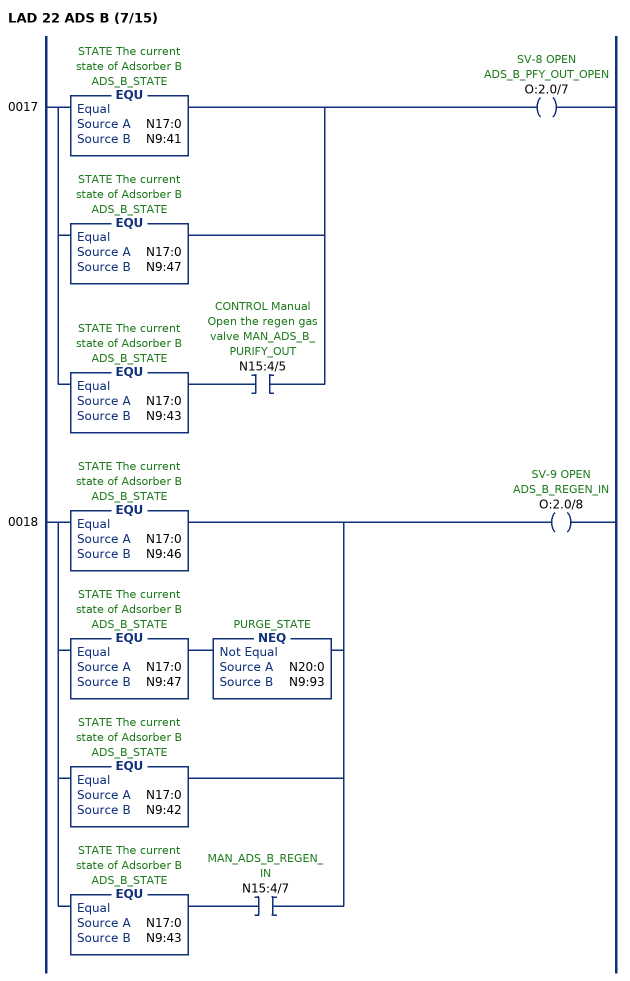
% Rung: 17 %
SOR BST EQU N17:0 N9:41 NXB EQU N17:0 N9:47 NXB EQU N17:0 N9:43 XIC N15:4/5 BND OTE O:2.0/7 EOR
%   N17:0  ADS_B_STATE  "STATE The current state of Adsorber B" %
%   N9:41  ADS_PURIFY  "STATE ADS Purify" %
%   N9:47  ADS_BACKFILL %
%   N9:43  ADS_MANUAL  "STATE ADS Manual" %
%   N15:4/5  MAN_ADS_B_PURIFY_OUT  "CONTROL Manual Open the regen gas valve" %
%   O:2.0/7  ADS_B_PFY_OUT_OPEN  "SV-8 OPEN" %
% Rung: 18 %
SOR BST EQU N17:0 N9:46 NXB EQU N17:0 N9:47 NEQ N20:0 N9:93 NXB EQU N17:0 N9:42 NXB EQU N17:0 N9:43 XIC N15:4/7 BND OTE O:2.0/8 EOR
%   N17:0  ADS_B_STATE  "STATE The current state of Adsorber B" %
%   N9:46  ADS_REGEN_BACKFILL %
%   N9:47  ADS_BACKFILL %
%   N20:0  PURGE_STATE %
%   N9:93  PURGE_BACKFILL %
%   N9:42  ADS_REGEN  "STATE ADS Regen" %
%   N9:43  ADS_MANUAL  "STATE ADS Manual" %
%   N15:4/7  MAN_ADS_B_REGEN_IN %
%   O:2.0/8  ADS_B_REGEN_IN  "SV-9 OPEN" %

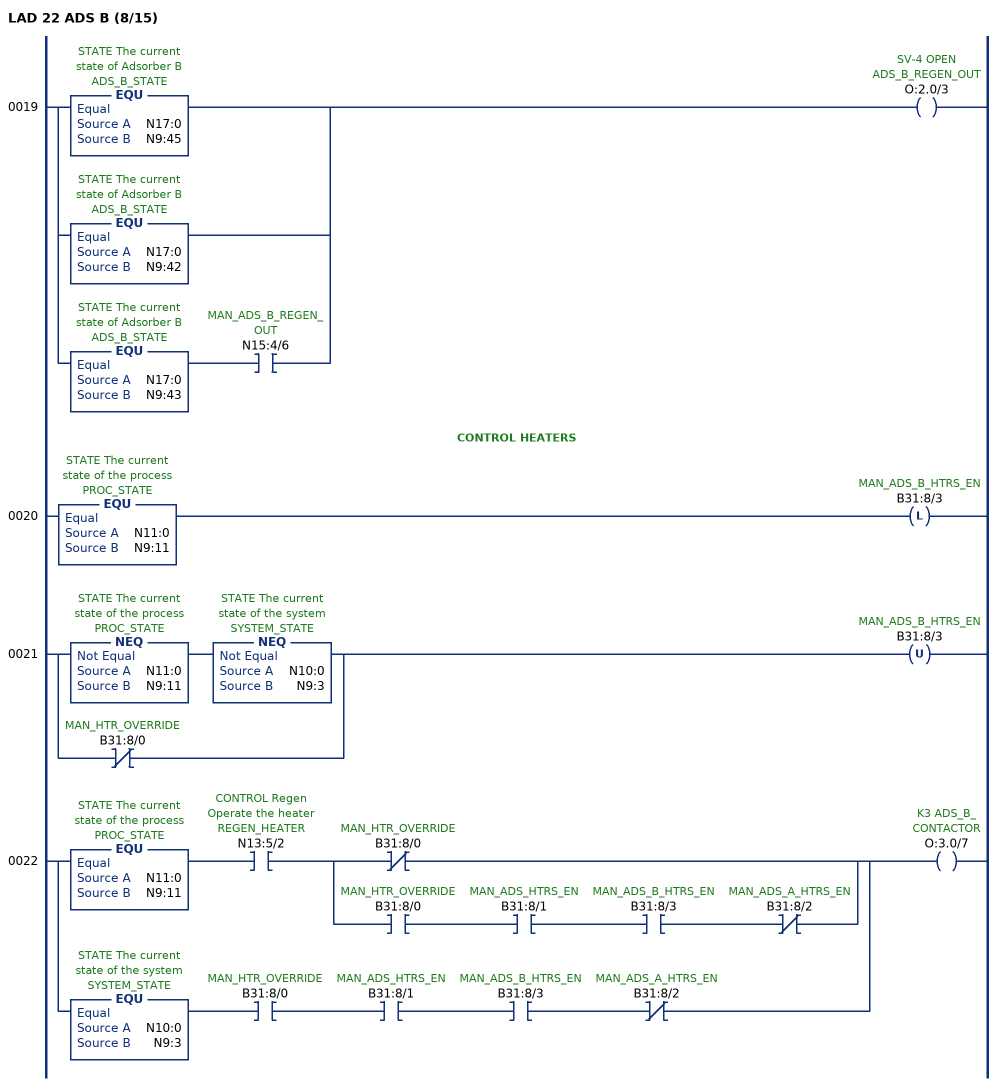
% Rung: 19 %
SOR BST EQU N17:0 N9:45 NXB EQU N17:0 N9:42 NXB EQU N17:0 N9:43 XIC N15:4/6 BND OTE O:2.0/3 EOR
%   N17:0  ADS_B_STATE  "STATE The current state of Adsorber B" %
%   N9:45  ADS_VENT %
%   N9:42  ADS_REGEN  "STATE ADS Regen" %
%   N9:43  ADS_MANUAL  "STATE ADS Manual" %
%   N15:4/6  MAN_ADS_B_REGEN_OUT %
%   O:2.0/3  ADS_B_REGEN_OUT  "SV-4 OPEN" %
% Rung: 20 %
% TITLE: CONTROL HEATERS %
SOR EQU N11:0 N9:11 OTL B31:8/3 EOR
%   N11:0  PROC_STATE  "STATE The current state of the process" %
%   N9:11  PROC_PFY_A_REG_B  "STATE Process Purify A" %
%   B31:8/3  MAN_ADS_B_HTRS_EN %
% Rung: 21 %
SOR BST NEQ N11:0 N9:11 NEQ N10:0 N9:3 NXB XIO B31:8/0 BND OTU B31:8/3 EOR
%   N11:0  PROC_STATE  "STATE The current state of the process" %
%   N9:11  PROC_PFY_A_REG_B  "STATE Process Purify A" %
%   N10:0  SYSTEM_STATE  "STATE The current state of the system" %
%   N9:3  SYSTEM_MANUAL  "STATE System Manual" %
%   B31:8/0  MAN_HTR_OVERRIDE %
%   B31:8/3  MAN_ADS_B_HTRS_EN %
% Rung: 22 %
SOR BST EQU N11:0 N9:11 XIC N13:5/2 BST XIO B31:8/0 NXB XIC B31:8/0 XIC B31:8/1 XIC B31:8/3 XIO B31:8/2 BND NXB EQU N10:0 N9:3 XIC B31:8/0 XIC B31:8/1 XIC B31:8/3 XIO B31:8/2 BND OTE O:3.0/7 EOR
%   N11:0  PROC_STATE  "STATE The current state of the process" %
%   N9:11  PROC_PFY_A_REG_B  "STATE Process Purify A" %
%   N13:5/2  REGEN_HEATER  "CONTROL Regen Operate the heater" %
%   B31:8/0  MAN_HTR_OVERRIDE %
%   B31:8/1  MAN_ADS_HTRS_EN %
%   B31:8/3  MAN_ADS_B_HTRS_EN %
%   B31:8/2  MAN_ADS_A_HTRS_EN %
%   N10:0  SYSTEM_STATE  "STATE The current state of the system" %
%   N9:3  SYSTEM_MANUAL  "STATE System Manual" %
%   O:3.0/7  ADS_B_CONTACTOR  "K3" %

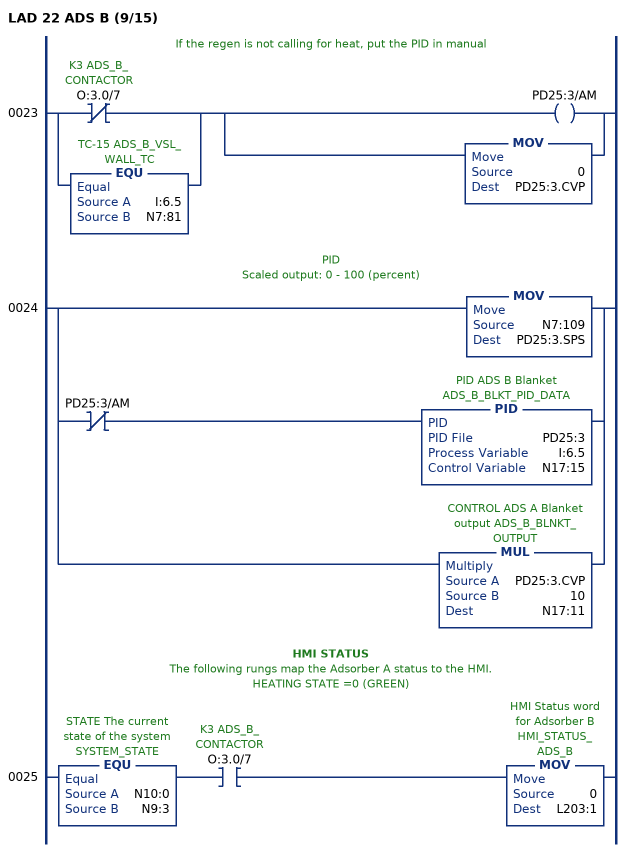
% Rung: 23 %
% If the regen is not calling for heat, put the PID in manual %
SOR BST XIO O:3.0/7 NXB EQU I:6.5 N7:81 BND BST OTE PD25:3/AM NXB MOV 0 PD25:3.CVP BND EOR
%   O:3.0/7  ADS_B_CONTACTOR  "K3" %
%   I:6.5  ADS_B_VSL_WALL_TC  "TC-15" %
%   N7:81  TC_OPEN_SP  "CONFIG The value read by an open TC input" %
% Rung: 24 %
% PID
% Scaled output: 0 - 100 (percent) %
SOR BST MOV N7:109 PD25:3.SPS NXB XIO PD25:3/AM PID PD25:3 I:6.5 N17:15 NXB MUL PD25:3.CVP 10 N17:11 BND EOR
%   N7:109  BLANKET_SP  "CONTROL Blanket PID Setpoint" %
%   PD25:3  ADS_B_BLKT_PID_DATA  "PID ADS B Blanket" %
%   I:6.5  ADS_B_VSL_WALL_TC  "TC-15" %
%   N17:15  ADS_B_BLKT_OUTPT_RAW  "CONTROL ADS B Blanket PID Output Raw" %
%   N17:11  ADS_B_BLNKT_OUTPUT  "CONTROL ADS A Blanket output" %
% Rung: 25 %
% TITLE: HMI STATUS %
% The following rungs map the Adsorber A status to the HMI.
% HEATING STATE =0 (GREEN) %
SOR EQU N10:0 N9:3 XIC O:3.0/7 MOV 0 L203:1 EOR
%   N10:0  SYSTEM_STATE  "STATE The current state of the system" %
%   N9:3  SYSTEM_MANUAL  "STATE System Manual" %
%   O:3.0/7  ADS_B_CONTACTOR  "K3" %
%   L203:1  HMI_STATUS_ADS_B  "HMI Status word for Adsorber B" %

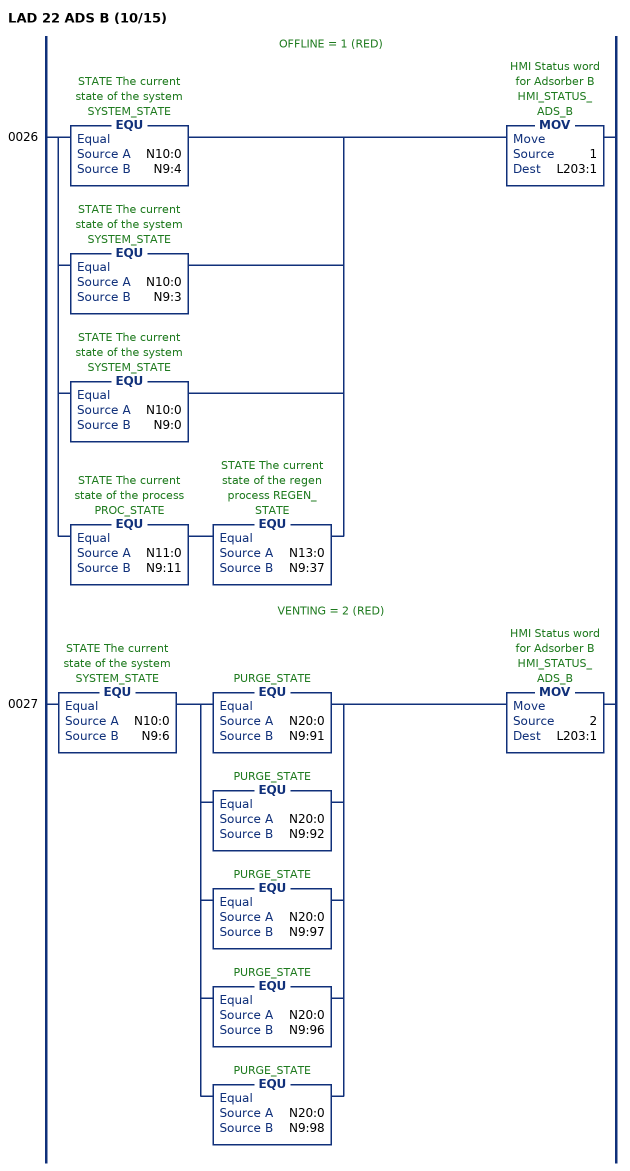
% Rung: 26 %
% OFFLINE = 1 (RED) %
SOR BST BST EQU N10:0 N9:4 NXB EQU N10:0 N9:3 NXB EQU N10:0 N9:0 BND NXB EQU N11:0 N9:11 EQU N13:0 N9:37 BND MOV 1 L203:1 EOR
%   N10:0  SYSTEM_STATE  "STATE The current state of the system" %
%   N9:4  SYSTEM_ALARM  "STATE System Alarm" %
%   N9:3  SYSTEM_MANUAL  "STATE System Manual" %
%   N9:0  SYSTEM_OFFLINE %
%   N11:0  PROC_STATE  "STATE The current state of the process" %
%   N9:11  PROC_PFY_A_REG_B  "STATE Process Purify A" %
%   N13:0  REGEN_STATE  "STATE The current state of the regen process" %
%   N9:37  REGEN_ALARM  "STATE Regen Alarm" %
%   L203:1  HMI_STATUS_ADS_B  "HMI Status word for Adsorber B" %
% Rung: 27 %
% VENTING = 2 (RED) %
SOR EQU N10:0 N9:6 BST EQU N20:0 N9:91 NXB EQU N20:0 N9:92 NXB EQU N20:0 N9:97 NXB EQU N20:0 N9:96 NXB EQU N20:0 N9:98 BND MOV 2 L203:1 EOR
%   N10:0  SYSTEM_STATE  "STATE The current state of the system" %
%   N9:6  SYSTEM_PURGE %
%   N20:0  PURGE_STATE %
%   N9:91  PURGE_INIT_VENT %
%   N9:92  PURGE_VENT_ADSORBER %
%   N9:97  PURGE_VENT_ADS_2 %
%   N9:96  PURGE_VENT_GETTER %
%   N9:98  PURGE_VENT_GET_2 %
%   L203:1  HMI_STATUS_ADS_B  "HMI Status word for Adsorber B" %

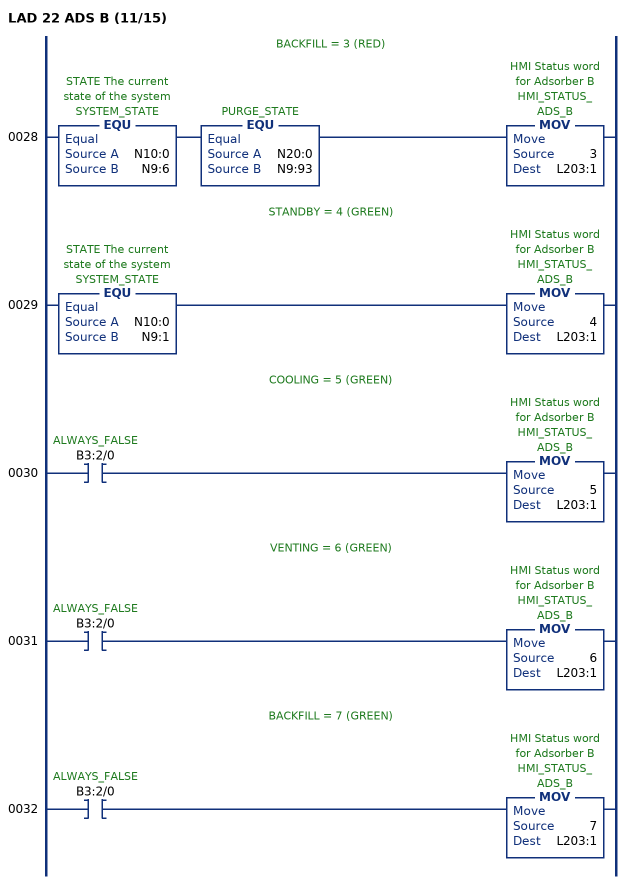
% Rung: 28 %
% BACKFILL = 3 (RED) %
SOR EQU N10:0 N9:6 EQU N20:0 N9:93 MOV 3 L203:1 EOR
%   N10:0  SYSTEM_STATE  "STATE The current state of the system" %
%   N9:6  SYSTEM_PURGE %
%   N20:0  PURGE_STATE %
%   N9:93  PURGE_BACKFILL %
%   L203:1  HMI_STATUS_ADS_B  "HMI Status word for Adsorber B" %
% Rung: 29 %
% STANDBY = 4 (GREEN) %
SOR EQU N10:0 N9:1 MOV 4 L203:1 EOR
%   N10:0  SYSTEM_STATE  "STATE The current state of the system" %
%   N9:1  SYSTEM_STANDBY  "STATE System Process" %
%   L203:1  HMI_STATUS_ADS_B  "HMI Status word for Adsorber B" %
% Rung: 30 %
% COOLING = 5 (GREEN) %
SOR XIC B3:2/0 MOV 5 L203:1 EOR
%   B3:2/0  ALWAYS_FALSE %
%   L203:1  HMI_STATUS_ADS_B  "HMI Status word for Adsorber B" %
% Rung: 31 %
% VENTING = 6 (GREEN) %
SOR XIC B3:2/0 MOV 6 L203:1 EOR
%   B3:2/0  ALWAYS_FALSE %
%   L203:1  HMI_STATUS_ADS_B  "HMI Status word for Adsorber B" %
% Rung: 32 %
% BACKFILL = 7 (GREEN) %
SOR XIC B3:2/0 MOV 7 L203:1 EOR
%   B3:2/0  ALWAYS_FALSE %
%   L203:1  HMI_STATUS_ADS_B  "HMI Status word for Adsorber B" %

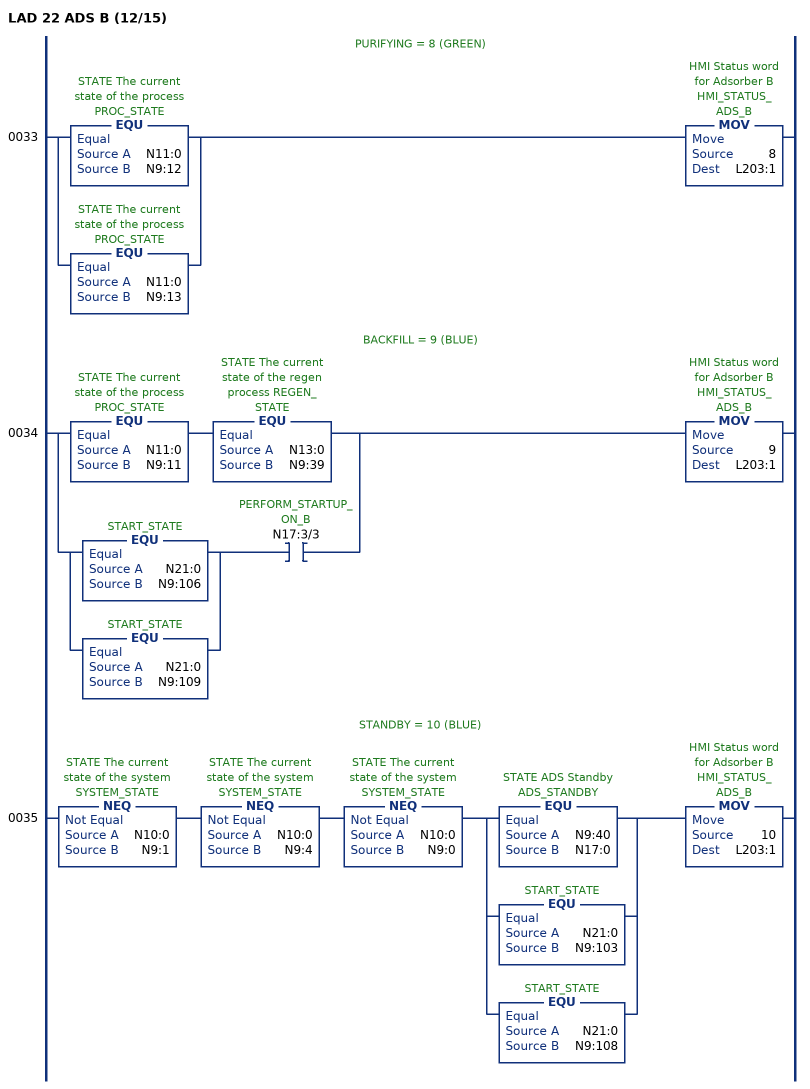
% Rung: 33 %
% PURIFYING = 8 (GREEN) %
SOR BST EQU N11:0 N9:12 NXB EQU N11:0 N9:13 BND MOV 8 L203:1 EOR
%   N11:0  PROC_STATE  "STATE The current state of the process" %
%   N9:12  PROC_PFY_B_REG_A  "STATE Process Purify B" %
%   N9:13  PROC_OVERLAP  "STATE Process Purify Overlap" %
%   L203:1  HMI_STATUS_ADS_B  "HMI Status word for Adsorber B" %
% Rung: 34 %
% BACKFILL = 9 (BLUE) %
SOR BST EQU N11:0 N9:11 EQU N13:0 N9:39 NXB BST EQU N21:0 N9:106 NXB EQU N21:0 N9:109 BND XIC N17:3/3 BND MOV 9 L203:1 EOR
%   N11:0  PROC_STATE  "STATE The current state of the process" %
%   N9:11  PROC_PFY_A_REG_B  "STATE Process Purify A" %
%   N13:0  REGEN_STATE  "STATE The current state of the regen process" %
%   N9:39  REGEN_BACKFILL %
%   N21:0  START_STATE %
%   N9:106  START_BACKFILL_1 %
%   N9:109  START_BKFL_2 %
%   N17:3/3  PERFORM_STARTUP_ON_B %
%   L203:1  HMI_STATUS_ADS_B  "HMI Status word for Adsorber B" %
% Rung: 35 %
% STANDBY = 10 (BLUE) %
SOR NEQ N10:0 N9:1 NEQ N10:0 N9:4 NEQ N10:0 N9:0 BST EQU N9:40 N17:0 NXB EQU N21:0 N9:103 NXB EQU N21:0 N9:108 BND MOV 10 L203:1 EOR
%   N10:0  SYSTEM_STATE  "STATE The current state of the system" %
%   N9:1  SYSTEM_STANDBY  "STATE System Process" %
%   N9:4  SYSTEM_ALARM  "STATE System Alarm" %
%   N9:0  SYSTEM_OFFLINE %
%   N9:40  ADS_STANDBY  "STATE ADS Standby" %
%   N17:0  ADS_B_STATE  "STATE The current state of Adsorber B" %
%   N21:0  START_STATE %
%   N9:103  START_VENT_GET_1 %
%   N9:108  START_VENT_GET_2 %
%   L203:1  HMI_STATUS_ADS_B  "HMI Status word for Adsorber B" %

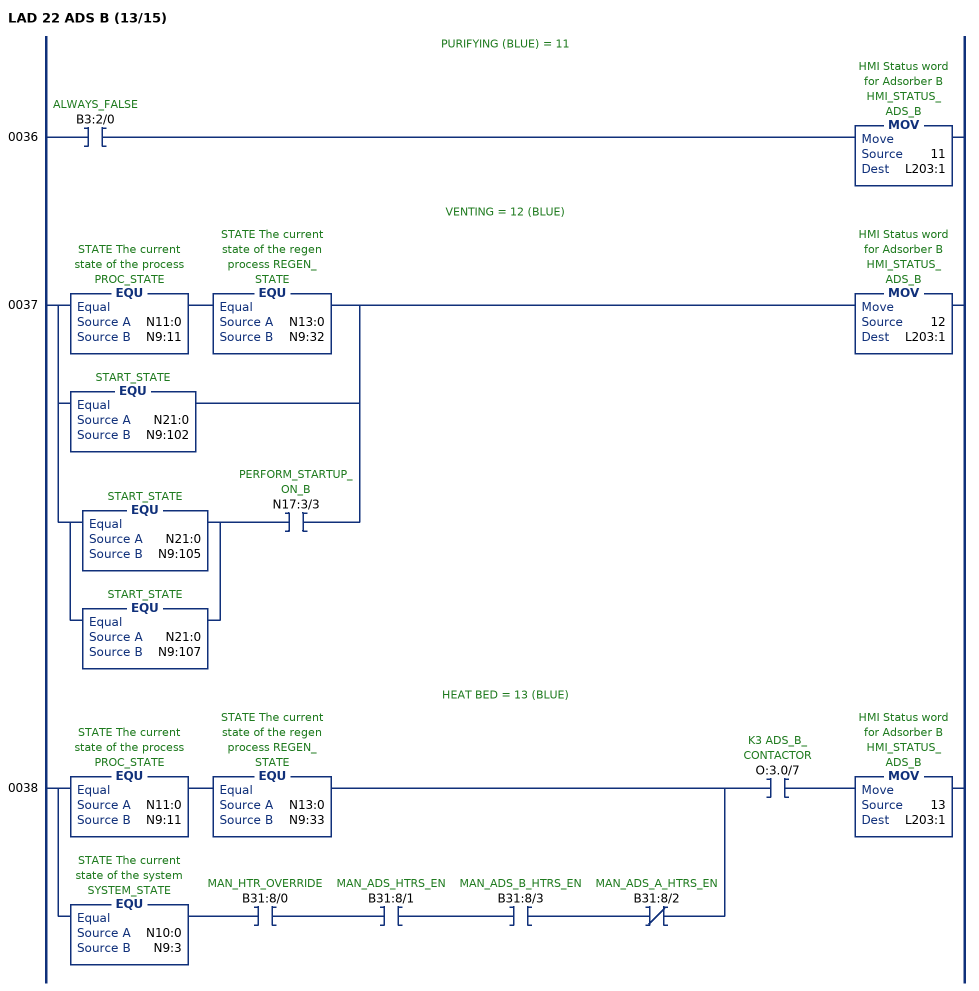
% Rung: 36 %
% PURIFYING (BLUE) = 11 %
SOR XIC B3:2/0 MOV 11 L203:1 EOR
%   B3:2/0  ALWAYS_FALSE %
%   L203:1  HMI_STATUS_ADS_B  "HMI Status word for Adsorber B" %
% Rung: 37 %
% VENTING = 12 (BLUE) %
SOR BST EQU N11:0 N9:11 EQU N13:0 N9:32 NXB BST EQU N21:0 N9:102 NXB BST EQU N21:0 N9:105 NXB EQU N21:0 N9:107 BND XIC N17:3/3 BND BND MOV 12 L203:1 EOR
%   N11:0  PROC_STATE  "STATE The current state of the process" %
%   N9:11  PROC_PFY_A_REG_B  "STATE Process Purify A" %
%   N13:0  REGEN_STATE  "STATE The current state of the regen process" %
%   N9:32  REGEN_VENT  "STATE Regen Vent" %
%   N21:0  START_STATE %
%   N9:102  START_VENT_ADS_1 %
%   N9:105  START_VENT_ALL %
%   N9:107  START_VENT_ADS_2 %
%   N17:3/3  PERFORM_STARTUP_ON_B %
%   L203:1  HMI_STATUS_ADS_B  "HMI Status word for Adsorber B" %
% Rung: 38 %
% HEAT BED = 13 (BLUE) %
SOR BST EQU N11:0 N9:11 EQU N13:0 N9:33 NXB EQU N10:0 N9:3 XIC B31:8/0 XIC B31:8/1 XIC B31:8/3 XIO B31:8/2 BND XIC O:3.0/7 MOV 13 L203:1 EOR
%   N11:0  PROC_STATE  "STATE The current state of the process" %
%   N9:11  PROC_PFY_A_REG_B  "STATE Process Purify A" %
%   N13:0  REGEN_STATE  "STATE The current state of the regen process" %
%   N9:33  REGEN_HEAT_BED  "STATE Regen Heat wall" %
%   N10:0  SYSTEM_STATE  "STATE The current state of the system" %
%   N9:3  SYSTEM_MANUAL  "STATE System Manual" %
%   B31:8/0  MAN_HTR_OVERRIDE %
%   B31:8/1  MAN_ADS_HTRS_EN %
%   B31:8/3  MAN_ADS_B_HTRS_EN %
%   B31:8/2  MAN_ADS_A_HTRS_EN %
%   O:3.0/7  ADS_B_CONTACTOR  "K3" %
%   L203:1  HMI_STATUS_ADS_B  "HMI Status word for Adsorber B" %

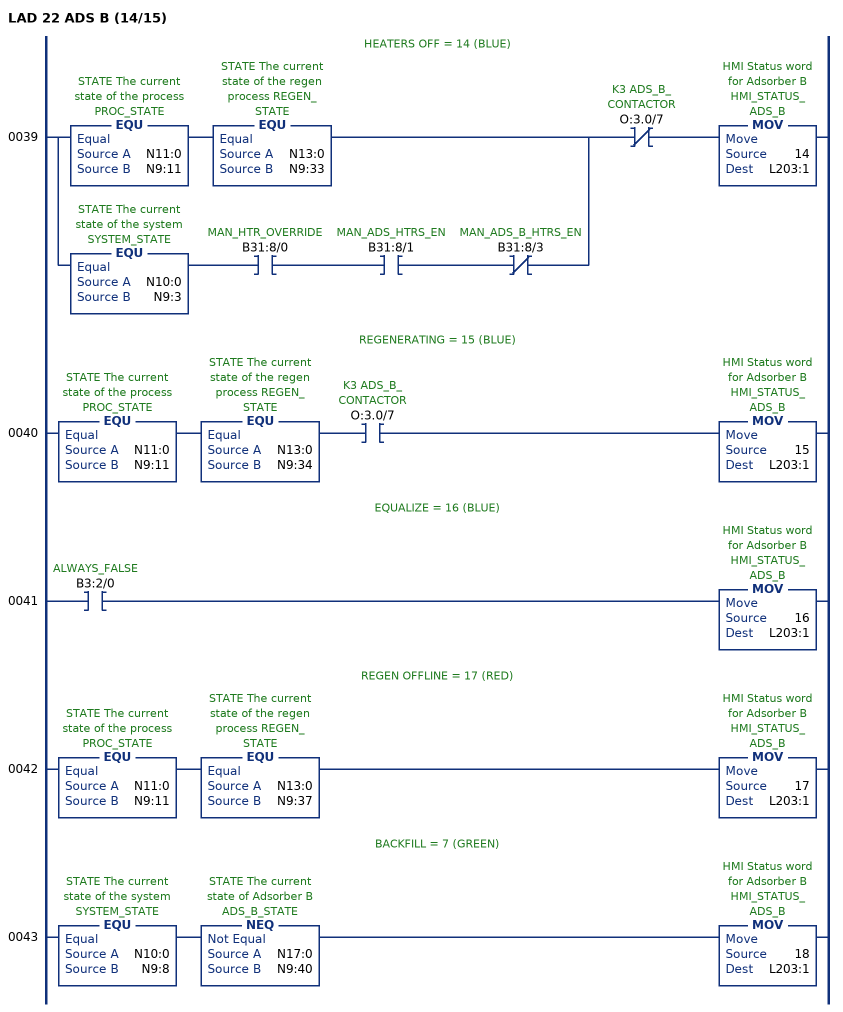
% Rung: 39 %
% HEATERS OFF = 14 (BLUE) %
SOR BST EQU N11:0 N9:11 EQU N13:0 N9:33 NXB EQU N10:0 N9:3 XIC B31:8/0 XIC B31:8/1 XIO B31:8/3 BND XIO O:3.0/7 MOV 14 L203:1 EOR
%   N11:0  PROC_STATE  "STATE The current state of the process" %
%   N9:11  PROC_PFY_A_REG_B  "STATE Process Purify A" %
%   N13:0  REGEN_STATE  "STATE The current state of the regen process" %
%   N9:33  REGEN_HEAT_BED  "STATE Regen Heat wall" %
%   N10:0  SYSTEM_STATE  "STATE The current state of the system" %
%   N9:3  SYSTEM_MANUAL  "STATE System Manual" %
%   B31:8/0  MAN_HTR_OVERRIDE %
%   B31:8/1  MAN_ADS_HTRS_EN %
%   B31:8/3  MAN_ADS_B_HTRS_EN %
%   O:3.0/7  ADS_B_CONTACTOR  "K3" %
%   L203:1  HMI_STATUS_ADS_B  "HMI Status word for Adsorber B" %
% Rung: 40 %
% REGENERATING = 15 (BLUE) %
SOR EQU N11:0 N9:11 EQU N13:0 N9:34 XIC O:3.0/7 MOV 15 L203:1 EOR
%   N11:0  PROC_STATE  "STATE The current state of the process" %
%   N9:11  PROC_PFY_A_REG_B  "STATE Process Purify A" %
%   N13:0  REGEN_STATE  "STATE The current state of the regen process" %
%   N9:34  REGEN_RUN  "STATE Regen Running" %
%   O:3.0/7  ADS_B_CONTACTOR  "K3" %
%   L203:1  HMI_STATUS_ADS_B  "HMI Status word for Adsorber B" %
% Rung: 41 %
% EQUALIZE = 16 (BLUE) %
SOR XIC B3:2/0 MOV 16 L203:1 EOR
%   B3:2/0  ALWAYS_FALSE %
%   L203:1  HMI_STATUS_ADS_B  "HMI Status word for Adsorber B" %
% Rung: 42 %
% REGEN OFFLINE = 17 (RED) %
SOR EQU N11:0 N9:11 EQU N13:0 N9:37 MOV 17 L203:1 EOR
%   N11:0  PROC_STATE  "STATE The current state of the process" %
%   N9:11  PROC_PFY_A_REG_B  "STATE Process Purify A" %
%   N13:0  REGEN_STATE  "STATE The current state of the regen process" %
%   N9:37  REGEN_ALARM  "STATE Regen Alarm" %
%   L203:1  HMI_STATUS_ADS_B  "HMI Status word for Adsorber B" %
% Rung: 43 %
% BACKFILL = 7 (GREEN) %
SOR EQU N10:0 N9:8 NEQ N17:0 N9:40 MOV 18 L203:1 EOR
%   N10:0  SYSTEM_STATE  "STATE The current state of the system" %
%   N9:8  SYSTEM_SUPPLEMENTAL %
%   N17:0  ADS_B_STATE  "STATE The current state of Adsorber B" %
%   N9:40  ADS_STANDBY  "STATE ADS Standby" %
%   L203:1  HMI_STATUS_ADS_B  "HMI Status word for Adsorber B" %

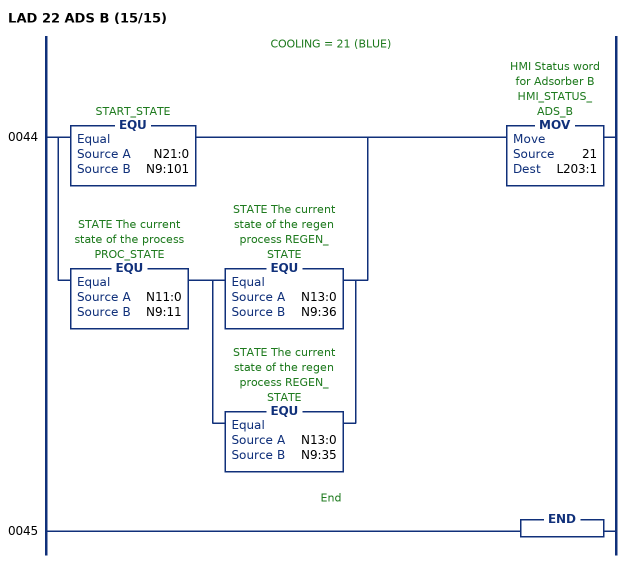
% Rung: 44 %
% COOLING = 21 (BLUE) %
SOR BST EQU N21:0 N9:101 NXB EQU N11:0 N9:11 BST EQU N13:0 N9:36 NXB EQU N13:0 N9:35 BND BND MOV 21 L203:1 EOR
%   N21:0  START_STATE %
%   N9:101  START_COOL %
%   N11:0  PROC_STATE  "STATE The current state of the process" %
%   N9:11  PROC_PFY_A_REG_B  "STATE Process Purify A" %
%   N13:0  REGEN_STATE  "STATE The current state of the regen process" %
%   N9:36  REGEN_COOL  "STATE Regen Cool" %
%   N9:35  REGEN_COOL_WALL  "STATE Regen Cool wall" %
%   L203:1  HMI_STATUS_ADS_B  "HMI Status word for Adsorber B" %
% Rung: 45 %
% End %
SOR END EOR

LADDER 23 "ADS B FLT"    % Controls the Adsorber B faults %
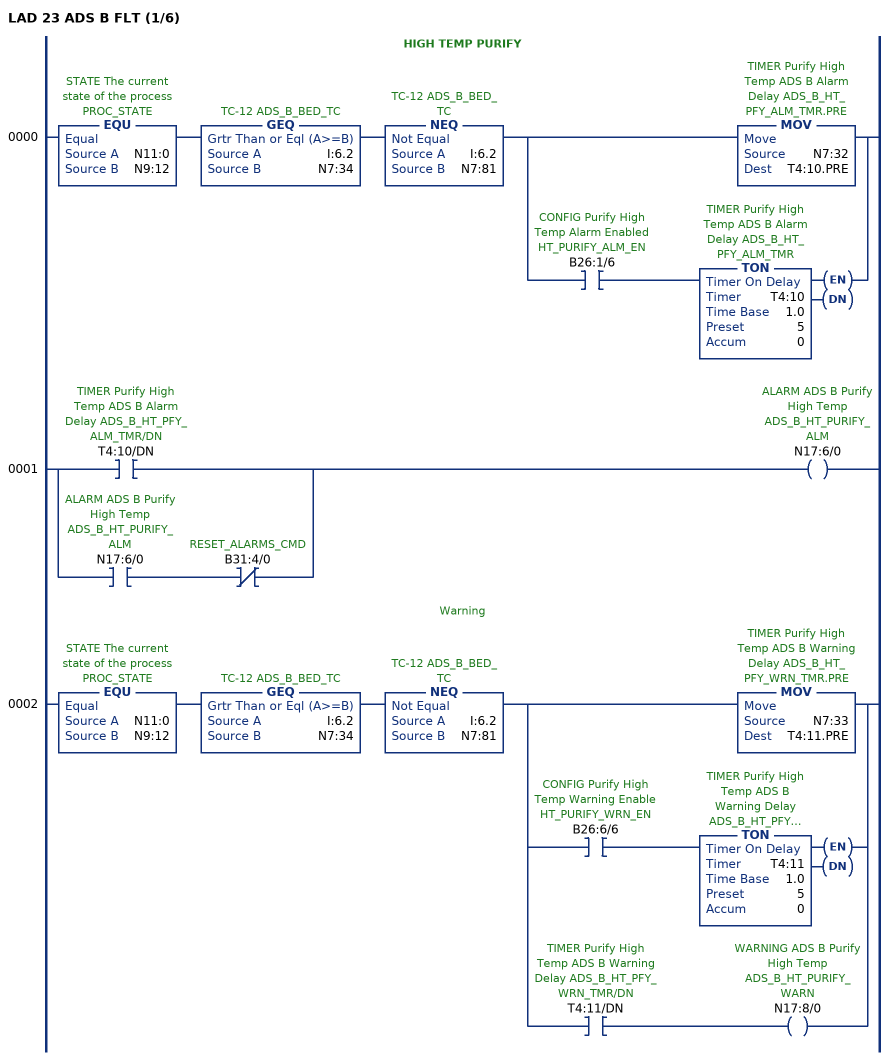
% Rung: 0 %
% TITLE: HIGH TEMP PURIFY %
SOR EQU N11:0 N9:12 GEQ I:6.2 N7:34 NEQ I:6.2 N7:81 BST MOV N7:32 T4:10.PRE NXB XIC B26:1/6 TON T4:10 1.0 5 0 BND EOR
%   N11:0  PROC_STATE  "STATE The current state of the process" %
%   N9:12  PROC_PFY_B_REG_A  "STATE Process Purify B" %
%   I:6.2  ADS_B_BED_TC  "TC-12" %
%   N7:34  HT_PURIFY_ALM_SP  "CONFIG Purify High Temp Alarm Setpoint" %
%   N7:81  TC_OPEN_SP  "CONFIG The value read by an open TC input" %
%   N7:32  HT_PURIFY_ALM_DLY  "CONFIG Purify High Temp Alarm Delay" %
%   T4:10  ADS_B_HT_PFY_ALM_TMR  "TIMER Purify High Temp ADS B Alarm Delay" %
%   B26:1/6  HT_PURIFY_ALM_EN  "CONFIG Purify High Temp Alarm Enabled" %
% Rung: 1 %
SOR BST XIC T4:10/DN NXB XIC N17:6/0 XIO B31:4/0 BND OTE N17:6/0 EOR
%   T4:10  ADS_B_HT_PFY_ALM_TMR  "TIMER Purify High Temp ADS B Alarm Delay" %
%   N17:6/0  ADS_B_HT_PURIFY_ALM  "ALARM ADS B Purify High Temp" %
%   B31:4/0  RESET_ALARMS_CMD %
% Rung: 2 %
% Warning %
SOR EQU N11:0 N9:12 GEQ I:6.2 N7:34 NEQ I:6.2 N7:81 BST MOV N7:33 T4:11.PRE NXB XIC B26:6/6 TON T4:11 1.0 5 0 NXB XIC T4:11/DN OTE N17:8/0 BND EOR
%   N11:0  PROC_STATE  "STATE The current state of the process" %
%   N9:12  PROC_PFY_B_REG_A  "STATE Process Purify B" %
%   I:6.2  ADS_B_BED_TC  "TC-12" %
%   N7:34  HT_PURIFY_ALM_SP  "CONFIG Purify High Temp Alarm Setpoint" %
%   N7:81  TC_OPEN_SP  "CONFIG The value read by an open TC input" %
%   N7:33  HT_PURIFY_WRN_DLY  "CONFIG Purify High Temp Warning Delay" %
%   T4:11  ADS_B_HT_PFY_WRN_TMR  "TIMER Purify High Temp ADS B Warning Delay" %
%   B26:6/6  HT_PURIFY_WRN_EN  "CONFIG Purify High Temp Warning Enable" %
%   N17:8/0  ADS_B_HT_PURIFY_WARN  "WARNING ADS B Purify High Temp" %

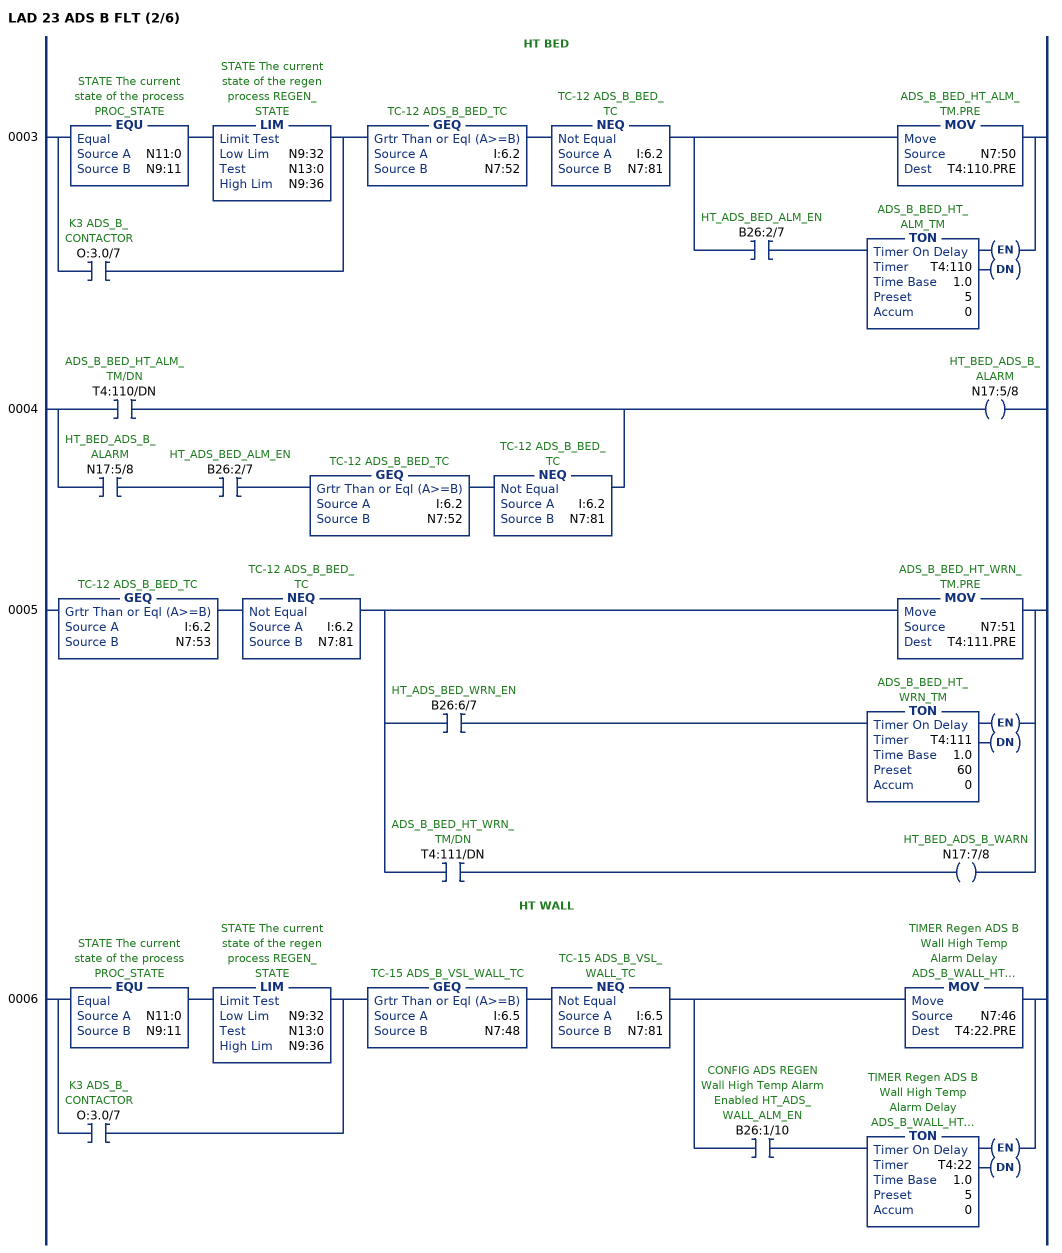
% Rung: 3 %
% TITLE: HT BED %
SOR BST EQU N11:0 N9:11 LIM N9:32 N13:0 N9:36 NXB XIC O:3.0/7 BND GEQ I:6.2 N7:52 NEQ I:6.2 N7:81 BST MOV N7:50 T4:110.PRE NXB XIC B26:2/7 TON T4:110 1.0 5 0 BND EOR
%   N11:0  PROC_STATE  "STATE The current state of the process" %
%   N9:11  PROC_PFY_A_REG_B  "STATE Process Purify A" %
%   N9:32  REGEN_VENT  "STATE Regen Vent" %
%   N13:0  REGEN_STATE  "STATE The current state of the regen process" %
%   N9:36  REGEN_COOL  "STATE Regen Cool" %
%   O:3.0/7  ADS_B_CONTACTOR  "K3" %
%   I:6.2  ADS_B_BED_TC  "TC-12" %
%   N7:52  HT_ADS_BED_ALM_SP %
%   N7:81  TC_OPEN_SP  "CONFIG The value read by an open TC input" %
%   N7:50  HT_ADS_BED_ALM_DLY %
%   T4:110  ADS_B_BED_HT_ALM_TM %
%   B26:2/7  HT_ADS_BED_ALM_EN %
% Rung: 4 %
SOR BST XIC T4:110/DN NXB XIC N17:5/8 XIC B26:2/7 GEQ I:6.2 N7:52 NEQ I:6.2 N7:81 BND OTE N17:5/8 EOR
%   T4:110  ADS_B_BED_HT_ALM_TM %
%   N17:5/8  HT_BED_ADS_B_ALARM %
%   B26:2/7  HT_ADS_BED_ALM_EN %
%   I:6.2  ADS_B_BED_TC  "TC-12" %
%   N7:52  HT_ADS_BED_ALM_SP %
%   N7:81  TC_OPEN_SP  "CONFIG The value read by an open TC input" %
% Rung: 5 %
SOR GEQ I:6.2 N7:53 NEQ I:6.2 N7:81 BST MOV N7:51 T4:111.PRE NXB XIC B26:6/7 TON T4:111 1.0 60 0 NXB XIC T4:111/DN OTE N17:7/8 BND EOR
%   I:6.2  ADS_B_BED_TC  "TC-12" %
%   N7:53  HT_ADS_BED_WRN_SP %
%   N7:81  TC_OPEN_SP  "CONFIG The value read by an open TC input" %
%   N7:51  HT_ADS_BED_WRN_DLY %
%   T4:111  ADS_B_BED_HT_WRN_TM %
%   B26:6/7  HT_ADS_BED_WRN_EN %
%   N17:7/8  HT_BED_ADS_B_WARN %
% Rung: 6 %
% TITLE: HT WALL %
SOR BST EQU N11:0 N9:11 LIM N9:32 N13:0 N9:36 NXB XIC O:3.0/7 BND GEQ I:6.5 N7:48 NEQ I:6.5 N7:81 BST MOV N7:46 T4:22.PRE NXB XIC B26:1/10 TON T4:22 1.0 5 0 BND EOR
%   N11:0  PROC_STATE  "STATE The current state of the process" %
%   N9:11  PROC_PFY_A_REG_B  "STATE Process Purify A" %
%   N9:32  REGEN_VENT  "STATE Regen Vent" %
%   N13:0  REGEN_STATE  "STATE The current state of the regen process" %
%   N9:36  REGEN_COOL  "STATE Regen Cool" %
%   O:3.0/7  ADS_B_CONTACTOR  "K3" %
%   I:6.5  ADS_B_VSL_WALL_TC  "TC-15" %
%   N7:48  HT_ADS_WALL_ALM_SP  "CONFIG ADS Wall Regen High Temp Alarm" %
%   N7:81  TC_OPEN_SP  "CONFIG The value read by an open TC input" %
%   N7:46  HT_ADS_WALL_ALM_DLY  "CONFIG ADS Wall High Temperature Alarm Delay" %
%   T4:22  ADS_B_WALL_HT_ALM_TM  "TIMER Regen ADS B Wall High Temp Alarm Delay" %
%   B26:1/10  HT_ADS_WALL_ALM_EN  "CONFIG ADS REGEN Wall High Temp Alarm Enabled" %

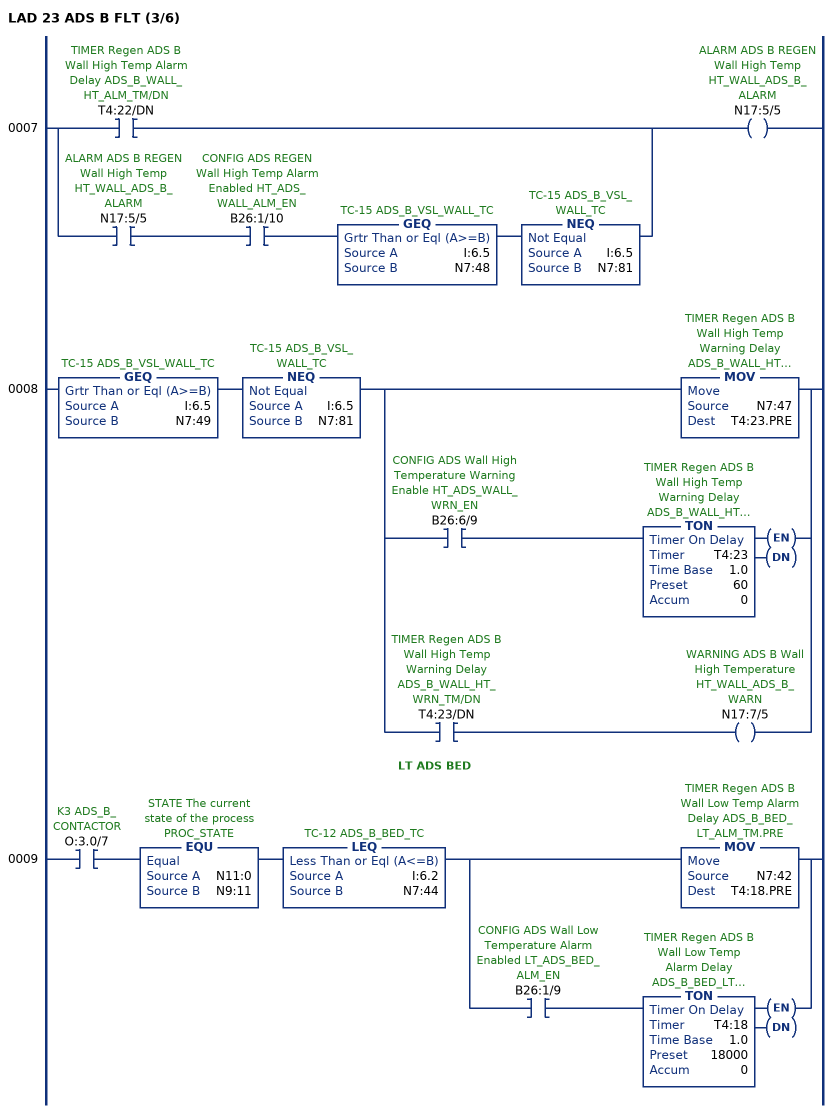
% Rung: 7 %
SOR BST XIC T4:22/DN NXB XIC N17:5/5 XIC B26:1/10 GEQ I:6.5 N7:48 NEQ I:6.5 N7:81 BND OTE N17:5/5 EOR
%   T4:22  ADS_B_WALL_HT_ALM_TM  "TIMER Regen ADS B Wall High Temp Alarm Delay" %
%   N17:5/5  HT_WALL_ADS_B_ALARM  "ALARM ADS B REGEN Wall High Temp" %
%   B26:1/10  HT_ADS_WALL_ALM_EN  "CONFIG ADS REGEN Wall High Temp Alarm Enabled" %
%   I:6.5  ADS_B_VSL_WALL_TC  "TC-15" %
%   N7:48  HT_ADS_WALL_ALM_SP  "CONFIG ADS Wall Regen High Temp Alarm" %
%   N7:81  TC_OPEN_SP  "CONFIG The value read by an open TC input" %
% Rung: 8 %
SOR GEQ I:6.5 N7:49 NEQ I:6.5 N7:81 BST MOV N7:47 T4:23.PRE NXB XIC B26:6/9 TON T4:23 1.0 60 0 NXB XIC T4:23/DN OTE N17:7/5 BND EOR
%   I:6.5  ADS_B_VSL_WALL_TC  "TC-15" %
%   N7:49  HT_ADS_WALL_WRN_SP  "CONFIG ADS Wall Regen High Temp Alarm" %
%   N7:81  TC_OPEN_SP  "CONFIG The value read by an open TC input" %
%   N7:47  HT_ADS_WALL_WRN_DLY  "CONFIG ADS Wall High Temperature Warning Delay" %
%   T4:23  ADS_B_WALL_HT_WRN_TM  "TIMER Regen ADS B Wall High Temp Warning Delay" %
%   B26:6/9  HT_ADS_WALL_WRN_EN  "CONFIG ADS Wall High Temperature Warning Enable" %
%   N17:7/5  HT_WALL_ADS_B_WARN  "WARNING ADS B Wall High Temperature" %
% Rung: 9 %
% TITLE: LT ADS BED %
SOR XIC O:3.0/7 EQU N11:0 N9:11 LEQ I:6.2 N7:44 BST MOV N7:42 T4:18.PRE NXB XIC B26:1/9 TON T4:18 1.0 18000 0 BND EOR
%   O:3.0/7  ADS_B_CONTACTOR  "K3" %
%   N11:0  PROC_STATE  "STATE The current state of the process" %
%   N9:11  PROC_PFY_A_REG_B  "STATE Process Purify A" %
%   I:6.2  ADS_B_BED_TC  "TC-12" %
%   N7:44  LT_ADS_BED_ALM_SP  "CONFIG ADS Wall Regen Heat Low Temperature Alarm Setpoint" %
%   N7:42  LT_ADS_BED_ALM_DLY  "CONFIG ADS Wall Regen heat Low Temperature Alarm Delay" %
%   T4:18  ADS_B_BED_LT_ALM_TM  "TIMER Regen ADS B Wall Low Temp Alarm Delay" %
%   B26:1/9  LT_ADS_BED_ALM_EN  "CONFIG ADS Wall Low Temperature Alarm Enabled" %

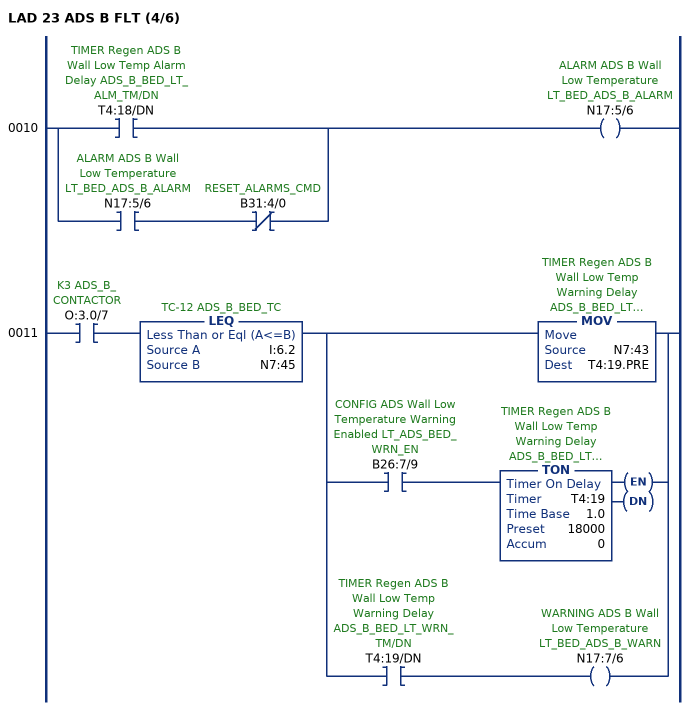
% Rung: 10 %
SOR BST XIC T4:18/DN NXB XIC N17:5/6 XIO B31:4/0 BND OTE N17:5/6 EOR
%   T4:18  ADS_B_BED_LT_ALM_TM  "TIMER Regen ADS B Wall Low Temp Alarm Delay" %
%   N17:5/6  LT_BED_ADS_B_ALARM  "ALARM ADS B Wall Low Temperature" %
%   B31:4/0  RESET_ALARMS_CMD %
% Rung: 11 %
SOR XIC O:3.0/7 LEQ I:6.2 N7:45 BST MOV N7:43 T4:19.PRE NXB XIC B26:7/9 TON T4:19 1.0 18000 0 NXB XIC T4:19/DN OTE N17:7/6 BND EOR
%   O:3.0/7  ADS_B_CONTACTOR  "K3" %
%   I:6.2  ADS_B_BED_TC  "TC-12" %
%   N7:45  LT_ADS_BED_WRN_SP  "CONFIG ADS Wall Regen Heat Low Temperature Warning Setpoint" %
%   N7:43  LT_ADS_BED_WRN_DLY  "CONFIG ADS Wall Regen heat Low Temperature Warning Delay" %
%   T4:19  ADS_B_BED_LT_WRN_TM  "TIMER Regen ADS B Wall Low Temp Warning Delay" %
%   B26:7/9  LT_ADS_BED_WRN_EN  "CONFIG ADS Wall Low Temperature Warning Enabled" %
%   N17:7/6  LT_BED_ADS_B_WARN  "WARNING ADS B Wall Low Temperature" %

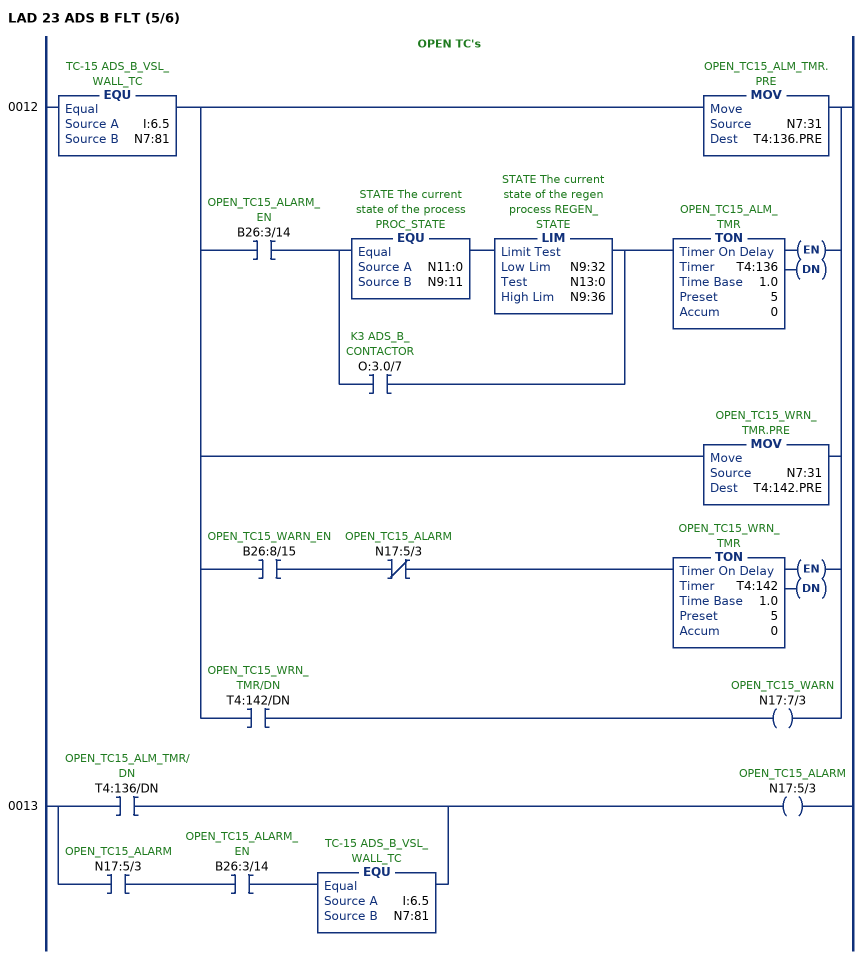
% Rung: 12 %
% TITLE: OPEN TC's %
SOR EQU I:6.5 N7:81 BST MOV N7:31 T4:136.PRE NXB XIC B26:3/14 BST EQU N11:0 N9:11 LIM N9:32 N13:0 N9:36 NXB XIC O:3.0/7 BND TON T4:136 1.0 5 0 NXB MOV N7:31 T4:142.PRE NXB XIC B26:8/15 XIO N17:5/3 TON T4:142 1.0 5 0 NXB XIC T4:142/DN OTE N17:7/3 BND EOR
%   I:6.5  ADS_B_VSL_WALL_TC  "TC-15" %
%   N7:81  TC_OPEN_SP  "CONFIG The value read by an open TC input" %
%   N7:31  OPEN_TC_DLY %
%   T4:136  OPEN_TC15_ALM_TMR %
%   B26:3/14  OPEN_TC15_ALARM_EN %
%   N11:0  PROC_STATE  "STATE The current state of the process" %
%   N9:11  PROC_PFY_A_REG_B  "STATE Process Purify A" %
%   N9:32  REGEN_VENT  "STATE Regen Vent" %
%   N13:0  REGEN_STATE  "STATE The current state of the regen process" %
%   N9:36  REGEN_COOL  "STATE Regen Cool" %
%   O:3.0/7  ADS_B_CONTACTOR  "K3" %
%   T4:142  OPEN_TC15_WRN_TMR %
%   B26:8/15  OPEN_TC15_WARN_EN %
%   N17:5/3  OPEN_TC15_ALARM %
%   N17:7/3  OPEN_TC15_WARN %
% Rung: 13 %
SOR BST XIC T4:136/DN NXB XIC N17:5/3 XIC B26:3/14 EQU I:6.5 N7:81 BND OTE N17:5/3 EOR
%   T4:136  OPEN_TC15_ALM_TMR %
%   N17:5/3  OPEN_TC15_ALARM %
%   B26:3/14  OPEN_TC15_ALARM_EN %
%   I:6.5  ADS_B_VSL_WALL_TC  "TC-15" %
%   N7:81  TC_OPEN_SP  "CONFIG The value read by an open TC input" %

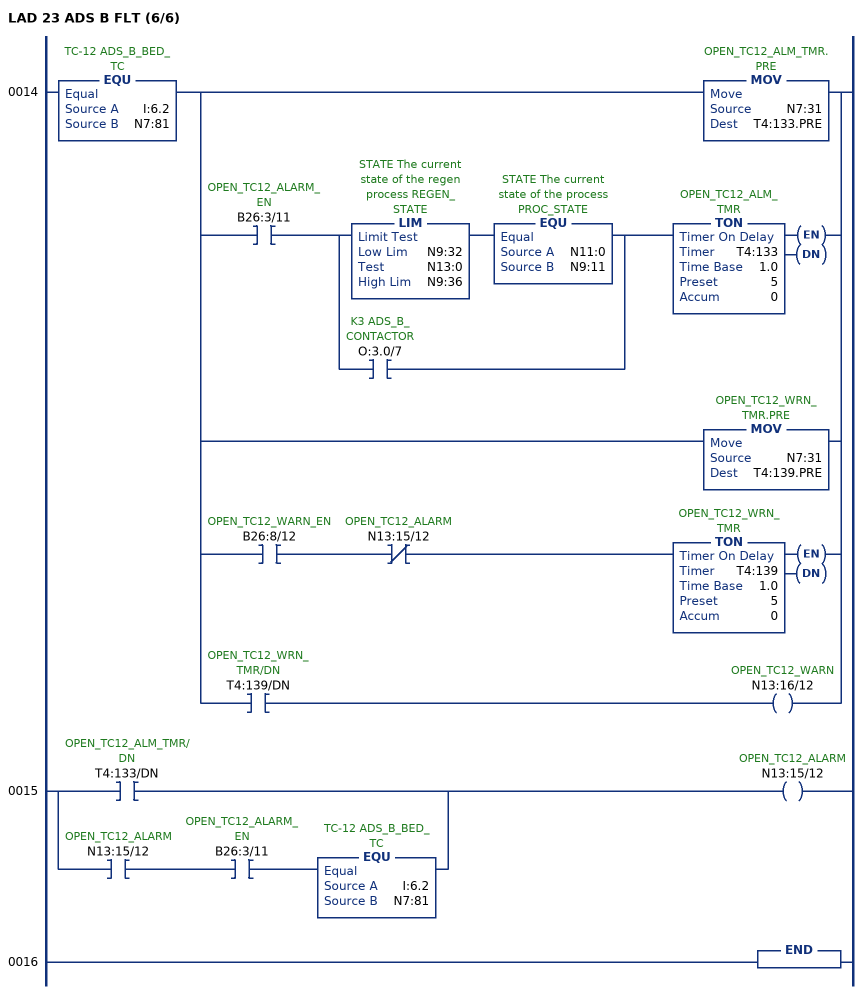
% Rung: 14 %
SOR EQU I:6.2 N7:81 BST MOV N7:31 T4:133.PRE NXB XIC B26:3/11 BST LIM N9:32 N13:0 N9:36 EQU N11:0 N9:11 NXB XIC O:3.0/7 BND TON T4:133 1.0 5 0 NXB MOV N7:31 T4:139.PRE NXB XIC B26:8/12 XIO N13:15/12 TON T4:139 1.0 5 0 NXB XIC T4:139/DN OTE N13:16/12 BND EOR
%   I:6.2  ADS_B_BED_TC  "TC-12" %
%   N7:81  TC_OPEN_SP  "CONFIG The value read by an open TC input" %
%   N7:31  OPEN_TC_DLY %
%   T4:133  OPEN_TC12_ALM_TMR %
%   B26:3/11  OPEN_TC12_ALARM_EN %
%   N9:32  REGEN_VENT  "STATE Regen Vent" %
%   N13:0  REGEN_STATE  "STATE The current state of the regen process" %
%   N9:36  REGEN_COOL  "STATE Regen Cool" %
%   N11:0  PROC_STATE  "STATE The current state of the process" %
%   N9:11  PROC_PFY_A_REG_B  "STATE Process Purify A" %
%   O:3.0/7  ADS_B_CONTACTOR  "K3" %
%   T4:139  OPEN_TC12_WRN_TMR %
%   B26:8/12  OPEN_TC12_WARN_EN %
%   N13:15/12  OPEN_TC12_ALARM %
%   N13:16/12  OPEN_TC12_WARN %
% Rung: 15 %
SOR BST XIC T4:133/DN NXB XIC N13:15/12 XIC B26:3/11 EQU I:6.2 N7:81 BND OTE N13:15/12 EOR
%   T4:133  OPEN_TC12_ALM_TMR %
%   N13:15/12  OPEN_TC12_ALARM %
%   B26:3/11  OPEN_TC12_ALARM_EN %
%   I:6.2  ADS_B_BED_TC  "TC-12" %
%   N7:81  TC_OPEN_SP  "CONFIG The value read by an open TC input" %
% Rung: 16 %
SOR END EOR

LADDER 24 "ADS PH"
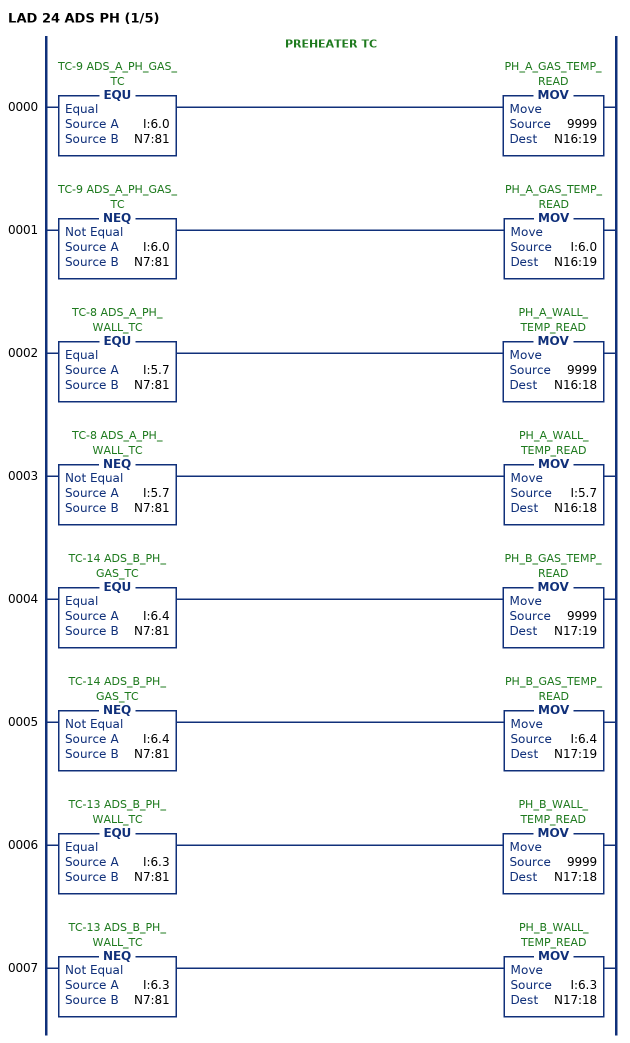
% Rung: 0 %
% TITLE: PREHEATER TC %
SOR EQU I:6.0 N7:81 MOV 9999 N16:19 EOR
%   I:6.0  ADS_A_PH_GAS_TC  "TC-9" %
%   N7:81  TC_OPEN_SP  "CONFIG The value read by an open TC input" %
%   N16:19  PH_A_GAS_TEMP_READ %
% Rung: 1 %
SOR NEQ I:6.0 N7:81 MOV I:6.0 N16:19 EOR
%   I:6.0  ADS_A_PH_GAS_TC  "TC-9" %
%   N7:81  TC_OPEN_SP  "CONFIG The value read by an open TC input" %
%   N16:19  PH_A_GAS_TEMP_READ %
% Rung: 2 %
SOR EQU I:5.7 N7:81 MOV 9999 N16:18 EOR
%   I:5.7  ADS_A_PH_WALL_TC  "TC-8" %
%   N7:81  TC_OPEN_SP  "CONFIG The value read by an open TC input" %
%   N16:18  PH_A_WALL_TEMP_READ %
% Rung: 3 %
SOR NEQ I:5.7 N7:81 MOV I:5.7 N16:18 EOR
%   I:5.7  ADS_A_PH_WALL_TC  "TC-8" %
%   N7:81  TC_OPEN_SP  "CONFIG The value read by an open TC input" %
%   N16:18  PH_A_WALL_TEMP_READ %
% Rung: 4 %
SOR EQU I:6.4 N7:81 MOV 9999 N17:19 EOR
%   I:6.4  ADS_B_PH_GAS_TC  "TC-14" %
%   N7:81  TC_OPEN_SP  "CONFIG The value read by an open TC input" %
%   N17:19  PH_B_GAS_TEMP_READ %
% Rung: 5 %
SOR NEQ I:6.4 N7:81 MOV I:6.4 N17:19 EOR
%   I:6.4  ADS_B_PH_GAS_TC  "TC-14" %
%   N7:81  TC_OPEN_SP  "CONFIG The value read by an open TC input" %
%   N17:19  PH_B_GAS_TEMP_READ %
% Rung: 6 %
SOR EQU I:6.3 N7:81 MOV 9999 N17:18 EOR
%   I:6.3  ADS_B_PH_WALL_TC  "TC-13" %
%   N7:81  TC_OPEN_SP  "CONFIG The value read by an open TC input" %
%   N17:18  PH_B_WALL_TEMP_READ %
% Rung: 7 %
SOR NEQ I:6.3 N7:81 MOV I:6.3 N17:18 EOR
%   I:6.3  ADS_B_PH_WALL_TC  "TC-13" %
%   N7:81  TC_OPEN_SP  "CONFIG The value read by an open TC input" %
%   N17:18  PH_B_WALL_TEMP_READ %

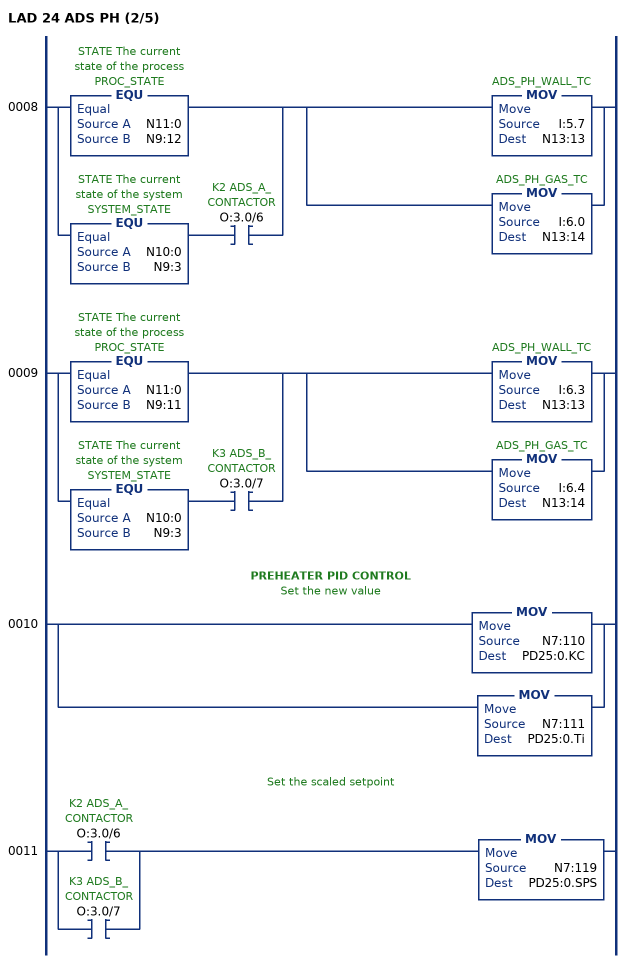
% Rung: 8 %
SOR BST EQU N11:0 N9:12 NXB EQU N10:0 N9:3 XIC O:3.0/6 BND BST MOV I:5.7 N13:13 NXB MOV I:6.0 N13:14 BND EOR
%   N11:0  PROC_STATE  "STATE The current state of the process" %
%   N9:12  PROC_PFY_B_REG_A  "STATE Process Purify B" %
%   N10:0  SYSTEM_STATE  "STATE The current state of the system" %
%   N9:3  SYSTEM_MANUAL  "STATE System Manual" %
%   O:3.0/6  ADS_A_CONTACTOR  "K2" %
%   I:5.7  ADS_A_PH_WALL_TC  "TC-8" %
%   N13:13  ADS_PH_WALL_TC %
%   I:6.0  ADS_A_PH_GAS_TC  "TC-9" %
%   N13:14  ADS_PH_GAS_TC %
% Rung: 9 %
SOR BST EQU N11:0 N9:11 NXB EQU N10:0 N9:3 XIC O:3.0/7 BND BST MOV I:6.3 N13:13 NXB MOV I:6.4 N13:14 BND EOR
%   N11:0  PROC_STATE  "STATE The current state of the process" %
%   N9:11  PROC_PFY_A_REG_B  "STATE Process Purify A" %
%   N10:0  SYSTEM_STATE  "STATE The current state of the system" %
%   N9:3  SYSTEM_MANUAL  "STATE System Manual" %
%   O:3.0/7  ADS_B_CONTACTOR  "K3" %
%   I:6.3  ADS_B_PH_WALL_TC  "TC-13" %
%   N13:13  ADS_PH_WALL_TC %
%   I:6.4  ADS_B_PH_GAS_TC  "TC-14" %
%   N13:14  ADS_PH_GAS_TC %
% Rung: 10 %
% TITLE: PREHEATER PID CONTROL %
% Set the new value %
SOR BST MOV N7:110 PD25:0.KC NXB MOV N7:111 PD25:0.Ti BND EOR
%   N7:110  PREHEATER_P  "CONFIG Preheater Proportional Gain New" %
%   N7:111  PREHEATER_I  "CONFIG Preheater Integral Gain New" %
% Rung: 11 %
% Set the scaled setpoint %
SOR BST XIC O:3.0/6 NXB XIC O:3.0/7 BND MOV N7:119 PD25:0.SPS EOR
%   O:3.0/6  ADS_A_CONTACTOR  "K2" %
%   O:3.0/7  ADS_B_CONTACTOR  "K3" %
%   N7:119  PREHEATER_SP  "CONTROL Preheater PID Setpoint" %

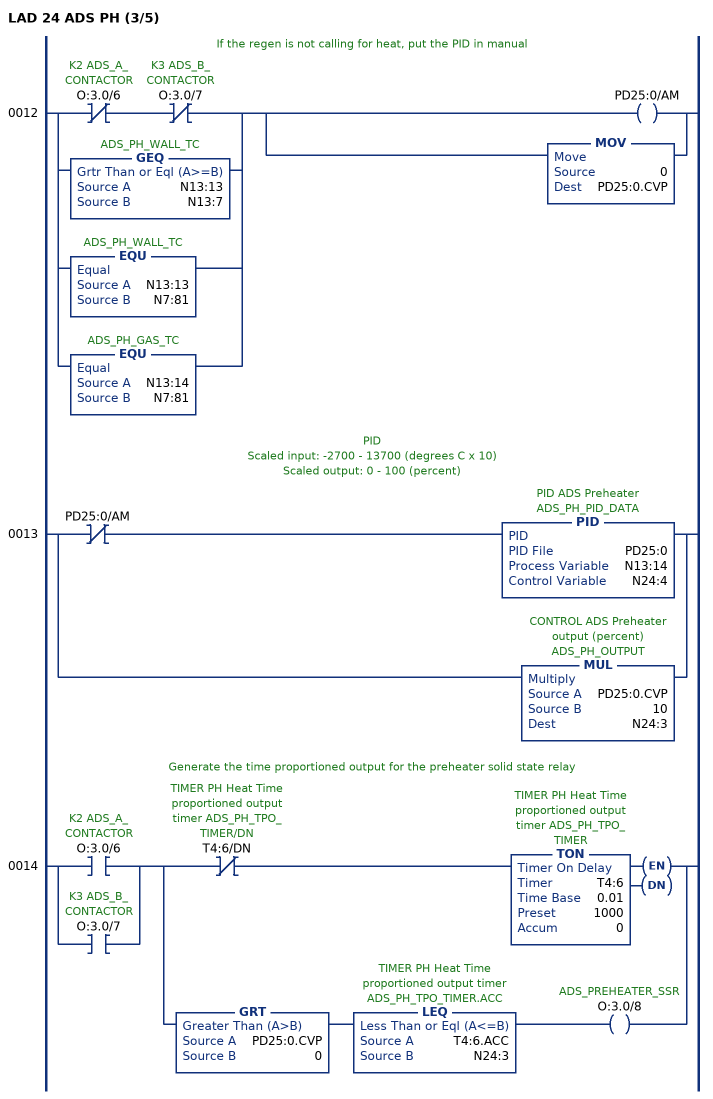
% Rung: 12 %
% If the regen is not calling for heat, put the PID in manual %
SOR BST XIO O:3.0/6 XIO O:3.0/7 NXB GEQ N13:13 N13:7 NXB EQU N13:13 N7:81 NXB EQU N13:14 N7:81 BND BST OTE PD25:0/AM NXB MOV 0 PD25:0.CVP BND EOR
%   O:3.0/6  ADS_A_CONTACTOR  "K2" %
%   O:3.0/7  ADS_B_CONTACTOR  "K3" %
%   N13:13  ADS_PH_WALL_TC %
%   N13:7  PH_WALL_LIMIT %
%   N7:81  TC_OPEN_SP  "CONFIG The value read by an open TC input" %
%   N13:14  ADS_PH_GAS_TC %
% Rung: 13 %
% PID
% Scaled input: -2700 - 13700 (degrees C x 10)
% Scaled output: 0 - 100 (percent) %
SOR BST XIO PD25:0/AM PID PD25:0 N13:14 N24:4 NXB MUL PD25:0.CVP 10 N24:3 BND EOR
%   PD25:0  ADS_PH_PID_DATA  "PID ADS Preheater" %
%   N13:14  ADS_PH_GAS_TC %
%   N24:4  ADS_PH_OUTPUT_RAW  "CONTROL ADS A Preheater PID Output Raw" %
%   N24:3  ADS_PH_OUTPUT  "CONTROL ADS Preheater output (percent)" %
% Rung: 14 %
% Generate the time proportioned output for the preheater solid state relay %
SOR BST XIC O:3.0/6 NXB XIC O:3.0/7 BND BST XIO T4:6/DN TON T4:6 0.01 1000 0 NXB GRT PD25:0.CVP 0 LEQ T4:6.ACC N24:3 OTE O:3.0/8 BND EOR
%   O:3.0/6  ADS_A_CONTACTOR  "K2" %
%   O:3.0/7  ADS_B_CONTACTOR  "K3" %
%   T4:6  ADS_PH_TPO_TIMER  "TIMER PH Heat Time proportioned output timer" %
%   N24:3  ADS_PH_OUTPUT  "CONTROL ADS Preheater output (percent)" %
%   O:3.0/8  ADS_PREHEATER_SSR %

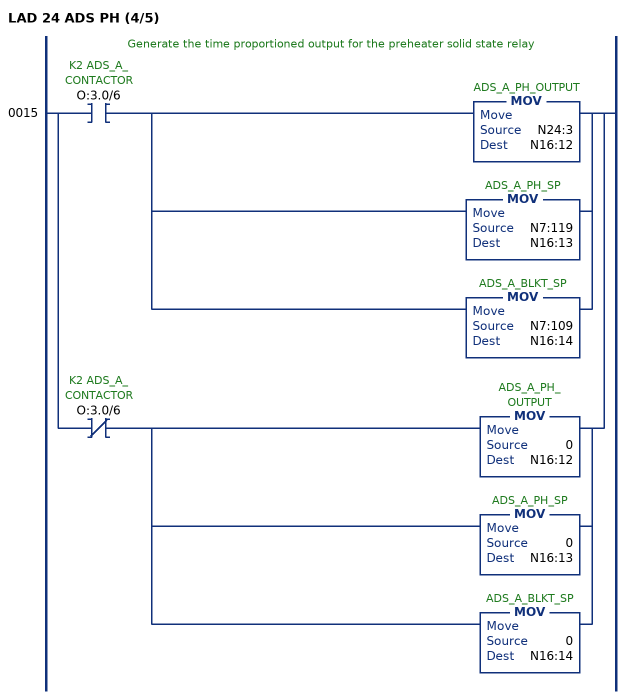
% Rung: 15 %
% Generate the time proportioned output for the preheater solid state relay %
SOR BST XIC O:3.0/6 BST MOV N24:3 N16:12 NXB MOV N7:119 N16:13 NXB MOV N7:109 N16:14 BND NXB XIO O:3.0/6 BST MOV 0 N16:12 NXB MOV 0 N16:13 NXB MOV 0 N16:14 BND BND EOR
%   O:3.0/6  ADS_A_CONTACTOR  "K2" %
%   N24:3  ADS_PH_OUTPUT  "CONTROL ADS Preheater output (percent)" %
%   N16:12  ADS_A_PH_OUTPUT %
%   N7:119  PREHEATER_SP  "CONTROL Preheater PID Setpoint" %
%   N16:13  ADS_A_PH_SP %
%   N7:109  BLANKET_SP  "CONTROL Blanket PID Setpoint" %
%   N16:14  ADS_A_BLKT_SP %

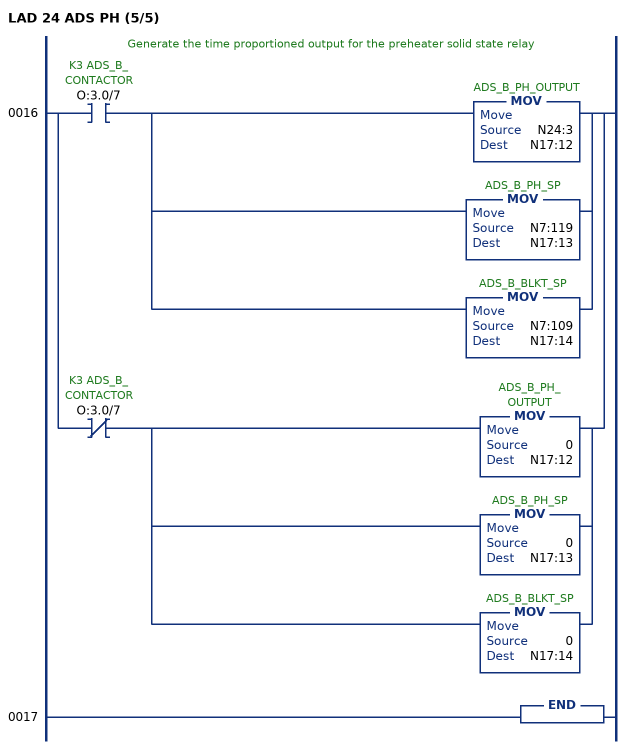
% Rung: 16 %
% Generate the time proportioned output for the preheater solid state relay %
SOR BST XIC O:3.0/7 BST MOV N24:3 N17:12 NXB MOV N7:119 N17:13 NXB MOV N7:109 N17:14 BND NXB XIO O:3.0/7 BST MOV 0 N17:12 NXB MOV 0 N17:13 NXB MOV 0 N17:14 BND BND EOR
%   O:3.0/7  ADS_B_CONTACTOR  "K3" %
%   N24:3  ADS_PH_OUTPUT  "CONTROL ADS Preheater output (percent)" %
%   N17:12  ADS_B_PH_OUTPUT %
%   N7:119  PREHEATER_SP  "CONTROL Preheater PID Setpoint" %
%   N17:13  ADS_B_PH_SP %
%   N7:109  BLANKET_SP  "CONTROL Blanket PID Setpoint" %
%   N17:14  ADS_B_BLKT_SP %
% Rung: 17 %
SOR END EOR

LADDER 25 "ADS PH FLT"
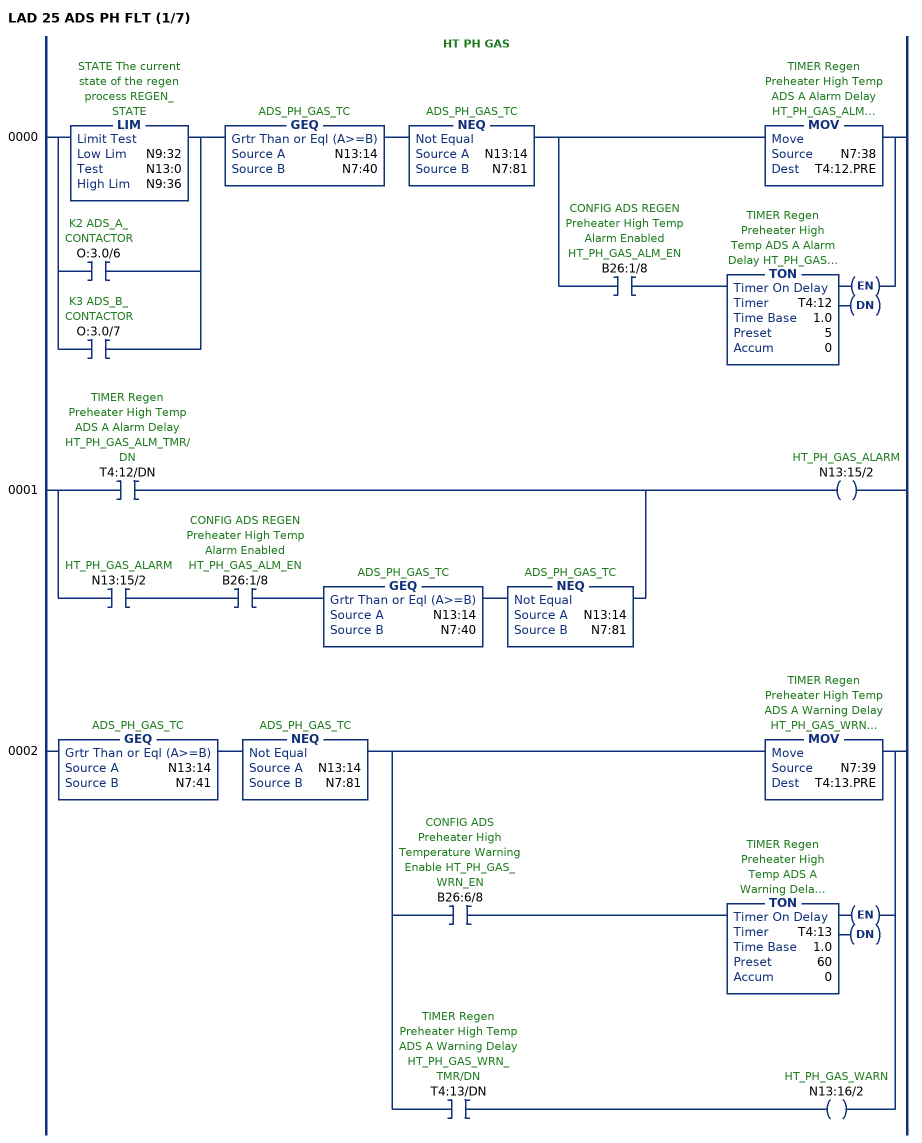
% Rung: 0 %
% TITLE: HT PH GAS %
SOR BST LIM N9:32 N13:0 N9:36 NXB XIC O:3.0/6 NXB XIC O:3.0/7 BND GEQ N13:14 N7:40 NEQ N13:14 N7:81 BST MOV N7:38 T4:12.PRE NXB XIC B26:1/8 TON T4:12 1.0 5 0 BND EOR
%   N9:32  REGEN_VENT  "STATE Regen Vent" %
%   N13:0  REGEN_STATE  "STATE The current state of the regen process" %
%   N9:36  REGEN_COOL  "STATE Regen Cool" %
%   O:3.0/6  ADS_A_CONTACTOR  "K2" %
%   O:3.0/7  ADS_B_CONTACTOR  "K3" %
%   N13:14  ADS_PH_GAS_TC %
%   N7:40  HT_PH_GAS_ALM_SP  "CONFIG ADS Preheater High Temperature Alarm Temperature" %
%   N7:81  TC_OPEN_SP  "CONFIG The value read by an open TC input" %
%   N7:38  HT_PH_GAS_ALM_DLY  "CONFIG ADS Preheater High Temperature Alarm Delay" %
%   T4:12  HT_PH_GAS_ALM_TMR  "TIMER Regen Preheater High Temp ADS A Alarm Delay" %
%   B26:1/8  HT_PH_GAS_ALM_EN  "CONFIG ADS REGEN Preheater High Temp Alarm Enabled" %
% Rung: 1 %
SOR BST XIC T4:12/DN NXB XIC N13:15/2 XIC B26:1/8 GEQ N13:14 N7:40 NEQ N13:14 N7:81 BND OTE N13:15/2 EOR
%   T4:12  HT_PH_GAS_ALM_TMR  "TIMER Regen Preheater High Temp ADS A Alarm Delay" %
%   N13:15/2  HT_PH_GAS_ALARM %
%   B26:1/8  HT_PH_GAS_ALM_EN  "CONFIG ADS REGEN Preheater High Temp Alarm Enabled" %
%   N13:14  ADS_PH_GAS_TC %
%   N7:40  HT_PH_GAS_ALM_SP  "CONFIG ADS Preheater High Temperature Alarm Temperature" %
%   N7:81  TC_OPEN_SP  "CONFIG The value read by an open TC input" %
% Rung: 2 %
SOR GEQ N13:14 N7:41 NEQ N13:14 N7:81 BST MOV N7:39 T4:13.PRE NXB XIC B26:6/8 TON T4:13 1.0 60 0 NXB XIC T4:13/DN OTE N13:16/2 BND EOR
%   N13:14  ADS_PH_GAS_TC %
%   N7:41  HT_PH_GAS_WRN_SP  "CONFIG ADS Preheater High Temperature Warning Temperature" %
%   N7:81  TC_OPEN_SP  "CONFIG The value read by an open TC input" %
%   N7:39  HT_PH_GAS_WRN_DLY  "CONFIG ADS Preheater High Temperature Warning Delay" %
%   T4:13  HT_PH_GAS_WRN_TMR  "TIMER Regen Preheater High Temp ADS A Warning Delay" %
%   B26:6/8  HT_PH_GAS_WRN_EN  "CONFIG ADS Preheater High Temperature Warning Enable" %
%   N13:16/2  HT_PH_GAS_WARN %

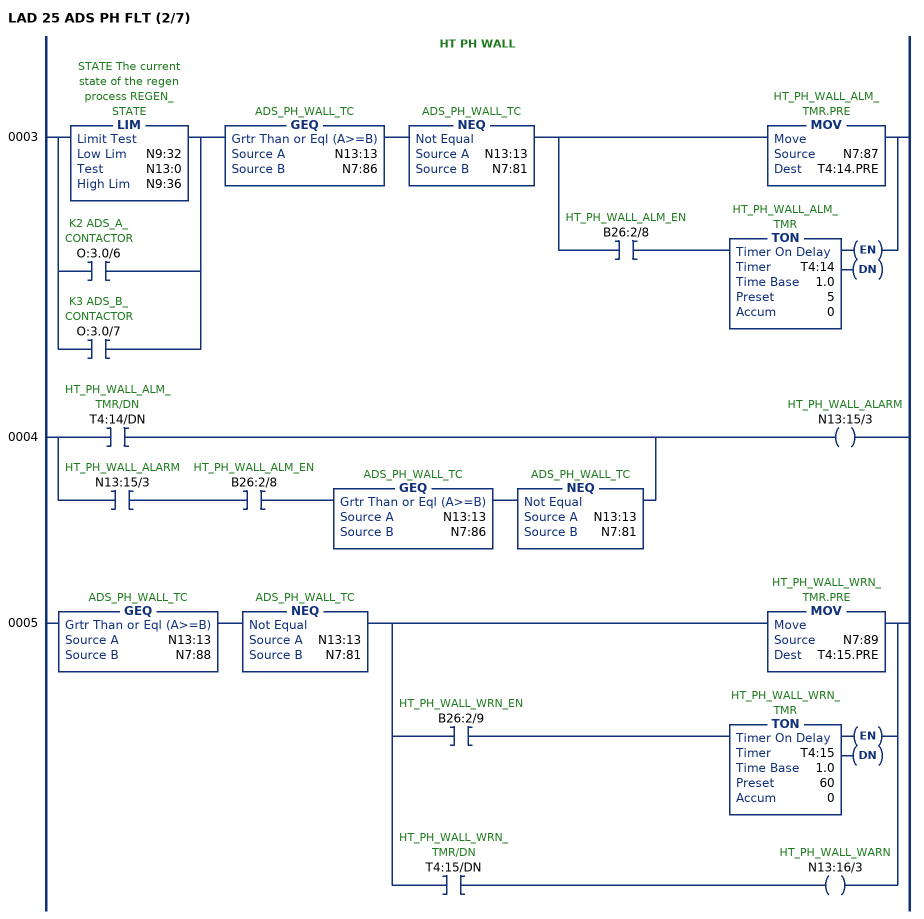
% Rung: 3 %
% TITLE: HT PH WALL %
SOR BST LIM N9:32 N13:0 N9:36 NXB XIC O:3.0/6 NXB XIC O:3.0/7 BND GEQ N13:13 N7:86 NEQ N13:13 N7:81 BST MOV N7:87 T4:14.PRE NXB XIC B26:2/8 TON T4:14 1.0 5 0 BND EOR
%   N9:32  REGEN_VENT  "STATE Regen Vent" %
%   N13:0  REGEN_STATE  "STATE The current state of the regen process" %
%   N9:36  REGEN_COOL  "STATE Regen Cool" %
%   O:3.0/6  ADS_A_CONTACTOR  "K2" %
%   O:3.0/7  ADS_B_CONTACTOR  "K3" %
%   N13:13  ADS_PH_WALL_TC %
%   N7:86  HT_PH_WALL_ALM_SP %
%   N7:81  TC_OPEN_SP  "CONFIG The value read by an open TC input" %
%   N7:87  HT_PH_WALL_ALM_DLY %
%   T4:14  HT_PH_WALL_ALM_TMR %
%   B26:2/8  HT_PH_WALL_ALM_EN %
% Rung: 4 %
SOR BST XIC T4:14/DN NXB XIC N13:15/3 XIC B26:2/8 GEQ N13:13 N7:86 NEQ N13:13 N7:81 BND OTE N13:15/3 EOR
%   T4:14  HT_PH_WALL_ALM_TMR %
%   N13:15/3  HT_PH_WALL_ALARM %
%   B26:2/8  HT_PH_WALL_ALM_EN %
%   N13:13  ADS_PH_WALL_TC %
%   N7:86  HT_PH_WALL_ALM_SP %
%   N7:81  TC_OPEN_SP  "CONFIG The value read by an open TC input" %
% Rung: 5 %
SOR GEQ N13:13 N7:88 NEQ N13:13 N7:81 BST MOV N7:89 T4:15.PRE NXB XIC B26:2/9 TON T4:15 1.0 60 0 NXB XIC T4:15/DN OTE N13:16/3 BND EOR
%   N13:13  ADS_PH_WALL_TC %
%   N7:88  HT_PH_WALL_WRN_SP %
%   N7:81  TC_OPEN_SP  "CONFIG The value read by an open TC input" %
%   N7:89  HT_PH_WALL_WRN_DLY %
%   T4:15  HT_PH_WALL_WRN_TMR %
%   B26:2/9  HT_PH_WALL_WRN_EN %
%   N13:16/3  HT_PH_WALL_WARN %

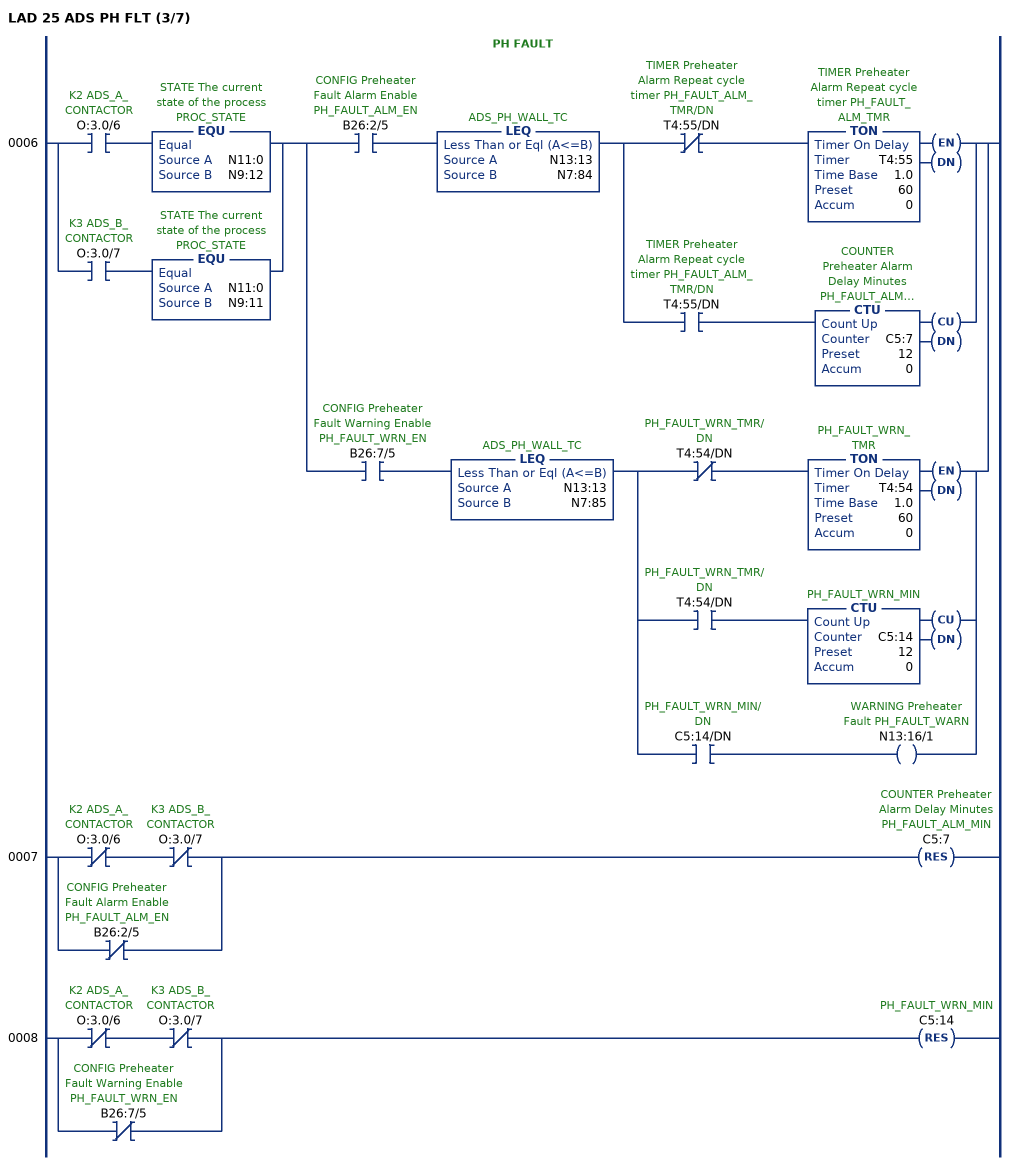
% Rung: 6 %
% TITLE: PH FAULT %
SOR BST XIC O:3.0/6 EQU N11:0 N9:12 NXB XIC O:3.0/7 EQU N11:0 N9:11 BND BST XIC B26:2/5 LEQ N13:13 N7:84 BST XIO T4:55/DN TON T4:55 1.0 60 0 NXB XIC T4:55/DN CTU C5:7 12 0 BND NXB XIC B26:7/5 LEQ N13:13 N7:85 BST XIO T4:54/DN TON T4:54 1.0 60 0 NXB XIC T4:54/DN CTU C5:14 12 0 NXB XIC C5:14/DN OTE N13:16/1 BND BND EOR
%   O:3.0/6  ADS_A_CONTACTOR  "K2" %
%   N11:0  PROC_STATE  "STATE The current state of the process" %
%   N9:12  PROC_PFY_B_REG_A  "STATE Process Purify B" %
%   O:3.0/7  ADS_B_CONTACTOR  "K3" %
%   N9:11  PROC_PFY_A_REG_B  "STATE Process Purify A" %
%   B26:2/5  PH_FAULT_ALM_EN  "CONFIG Preheater Fault Alarm Enable" %
%   N13:13  ADS_PH_WALL_TC %
%   N7:84  PH_FAULT_ALARM_SP  "CONFIG Preheater Temperature Delta Alarm Setpoint" %
%   T4:55  PH_FAULT_ALM_TMR  "TIMER Preheater Alarm Repeat cycle timer" %
%   C5:7  PH_FAULT_ALM_MIN  "COUNTER Preheater Alarm Delay Minutes" %
%   B26:7/5  PH_FAULT_WRN_EN  "CONFIG Preheater Fault Warning Enable" %
%   N7:85  PH_FAULT_WARN_SP %
%   T4:54  PH_FAULT_WRN_TMR %
%   C5:14  PH_FAULT_WRN_MIN %
%   N13:16/1  PH_FAULT_WARN  "WARNING Preheater Fault" %
% Rung: 7 %
SOR BST XIO O:3.0/6 XIO O:3.0/7 NXB XIO B26:2/5 BND RES C5:7 EOR
%   O:3.0/6  ADS_A_CONTACTOR  "K2" %
%   O:3.0/7  ADS_B_CONTACTOR  "K3" %
%   B26:2/5  PH_FAULT_ALM_EN  "CONFIG Preheater Fault Alarm Enable" %
%   C5:7  PH_FAULT_ALM_MIN  "COUNTER Preheater Alarm Delay Minutes" %
% Rung: 8 %
SOR BST XIO O:3.0/6 XIO O:3.0/7 NXB XIO B26:7/5 BND RES C5:14 EOR
%   O:3.0/6  ADS_A_CONTACTOR  "K2" %
%   O:3.0/7  ADS_B_CONTACTOR  "K3" %
%   B26:7/5  PH_FAULT_WRN_EN  "CONFIG Preheater Fault Warning Enable" %
%   C5:14  PH_FAULT_WRN_MIN %

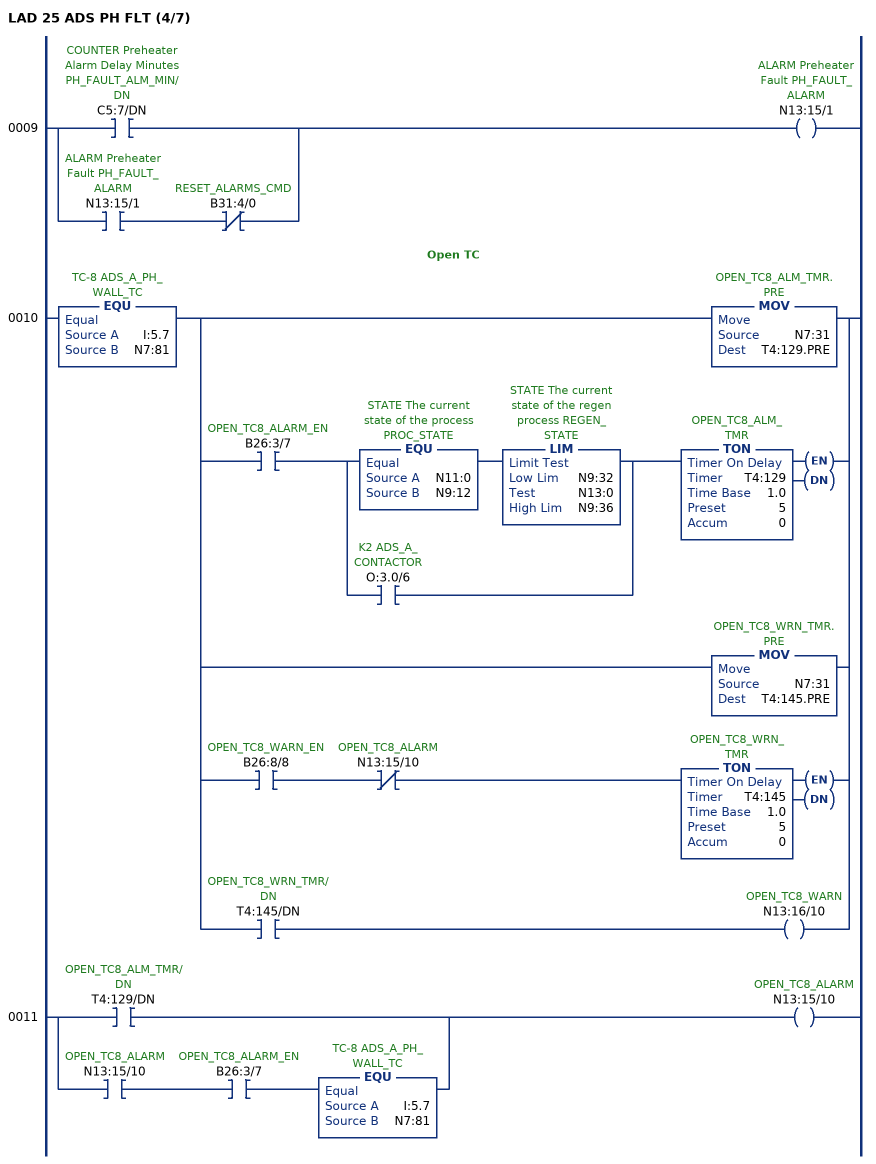
% Rung: 9 %
SOR BST XIC C5:7/DN NXB XIC N13:15/1 XIO B31:4/0 BND OTE N13:15/1 EOR
%   C5:7  PH_FAULT_ALM_MIN  "COUNTER Preheater Alarm Delay Minutes" %
%   N13:15/1  PH_FAULT_ALARM  "ALARM Preheater Fault" %
%   B31:4/0  RESET_ALARMS_CMD %
% Rung: 10 %
% TITLE: Open TC %
SOR EQU I:5.7 N7:81 BST MOV N7:31 T4:129.PRE NXB XIC B26:3/7 BST EQU N11:0 N9:12 LIM N9:32 N13:0 N9:36 NXB XIC O:3.0/6 BND TON T4:129 1.0 5 0 NXB MOV N7:31 T4:145.PRE NXB XIC B26:8/8 XIO N13:15/10 TON T4:145 1.0 5 0 NXB XIC T4:145/DN OTE N13:16/10 BND EOR
%   I:5.7  ADS_A_PH_WALL_TC  "TC-8" %
%   N7:81  TC_OPEN_SP  "CONFIG The value read by an open TC input" %
%   N7:31  OPEN_TC_DLY %
%   T4:129  OPEN_TC8_ALM_TMR %
%   B26:3/7  OPEN_TC8_ALARM_EN %
%   N11:0  PROC_STATE  "STATE The current state of the process" %
%   N9:12  PROC_PFY_B_REG_A  "STATE Process Purify B" %
%   N9:32  REGEN_VENT  "STATE Regen Vent" %
%   N13:0  REGEN_STATE  "STATE The current state of the regen process" %
%   N9:36  REGEN_COOL  "STATE Regen Cool" %
%   O:3.0/6  ADS_A_CONTACTOR  "K2" %
%   T4:145  OPEN_TC8_WRN_TMR %
%   B26:8/8  OPEN_TC8_WARN_EN %
%   N13:15/10  OPEN_TC8_ALARM %
%   N13:16/10  OPEN_TC8_WARN %
% Rung: 11 %
SOR BST XIC T4:129/DN NXB XIC N13:15/10 XIC B26:3/7 EQU I:5.7 N7:81 BND OTE N13:15/10 EOR
%   T4:129  OPEN_TC8_ALM_TMR %
%   N13:15/10  OPEN_TC8_ALARM %
%   B26:3/7  OPEN_TC8_ALARM_EN %
%   I:5.7  ADS_A_PH_WALL_TC  "TC-8" %
%   N7:81  TC_OPEN_SP  "CONFIG The value read by an open TC input" %

